// TIA Portal V20 export
FUNCTION_BLOCK "LER_DiagnosticsStatus"   // FB29, LAD
// stored: Access Published, MemoryReserve 100, SetENOAutomatically false
   VAR_INPUT
      devStateHmi_X1 : Array[0..256] of "LAF_typeDevDiagBasic";
      devStateHmi_X2 : Array[0..256] of "LAF_typeDevDiagBasic";
      UnitSelect : Int;
      Reset : Bool;
   END_VAR
   VAR_IN_OUT
      DevState : "LER_DiagnosticsInterface";
   END_VAR
   VAR
      staticCntState : Int := 1;
      staticCntStartState : Int := 1;
      staticCntEndState : Int := 200;
      staticCntDev : Int := 1;
      staticCntHighLimit_X2 : Array[1..15] of Int;
      staticCntLowLimit_X2 : Array[1..15] of Int;
      staticCntHighLimit_X1 : Array[1..15] of Int;
      staticCntLowLimit_X1 : Array[1..15] of Int;
      staticCntModuleState : Int;
      staticDevStateError : Array[0..15] of Bool;
      statiDevStateMove_X1 : Array[0..15] of Int;
      statiDevStateMove_X2 : Array[0..15] of Int;
   END_VAR
   VAR_TEMP
      tempIndex : Int;
   END_VAR
   VAR CONSTANT
      nomal : Word := 16#0009;
   END_VAR
   // staticCntHighLimit_X2[1] := 12;
   // staticCntHighLimit_X2[2] := 14;
   // staticCntHighLimit_X2[3] := 18;
   // staticCntHighLimit_X2[4] := 35;
   // staticCntHighLimit_X2[5] := 38;
   // staticCntHighLimit_X2[6] := 39;
   // staticCntHighLimit_X2[7] := 51;
   // staticCntHighLimit_X2[8] := 53;
   // staticCntLowLimit_X2[2] := 11;
   // staticCntLowLimit_X2[3] := 13;
   // staticCntLowLimit_X2[4] := 17;
   // staticCntLowLimit_X2[5] := 34;
   // staticCntLowLimit_X2[6] := 37;
   // staticCntLowLimit_X2[7] := 38;
   // staticCntLowLimit_X2[8] := 50;
   // staticCntHighLimit_X1[1] := 12;
   // staticCntHighLimit_X1[2] := 14;
   // staticCntHighLimit_X1[3] := 18;
   // staticCntHighLimit_X1[4] := 35;
   // staticCntHighLimit_X1[5] := 38;
   // staticCntHighLimit_X1[6] := 39;
   // staticCntHighLimit_X1[7] := 51;
   // staticCntHighLimit_X1[8] := 53;
   // staticCntLowLimit_X1[2] := 11;
   // staticCntLowLimit_X1[3] := 13;
   // staticCntLowLimit_X1[4] := 17;
   // staticCntLowLimit_X1[5] := 34;
   // staticCntLowLimit_X1[6] := 37;
   // staticCntLowLimit_X1[7] := 38;
   // staticCntLowLimit_X1[8] := 50;
   VAR_TEMP   // added for the SCL form of the ladder/FBD networks
      _w1 : Bool;
      _w2 : Bool;
      _w3 : Bool;
      _w4 : Bool;
      _w5 : Bool;
      _w6 : Bool;
      _w7 : Bool;
      _w8 : Bool;
      _w9 : Bool;
      _w10 : Bool;
      _w11 : Bool;
      _w12 : Bool;
      _w13 : Bool;
      _w14 : Bool;
      _w15 : Bool;
      _w16 : Bool;
   END_VAR
BEGIN

REGION Network 1 (SCL): X1 Port Range
   CASE #UnitSelect OF
       1:  // Unit Reelcut Anode
           #staticCntHighLimit_X1[1] := 0;
           #staticCntHighLimit_X1[2] := 0;
           #staticCntHighLimit_X1[3] := 0;
           #staticCntHighLimit_X1[4] := 18;
           #staticCntHighLimit_X1[5] := 0;
           #staticCntHighLimit_X1[6] := 0;
           #staticCntHighLimit_X1[7] := 41;
           #staticCntHighLimit_X1[8] := 0;
           #staticCntHighLimit_X1[9] := 0;
           #staticCntHighLimit_X1[10] := 0;
           #staticCntHighLimit_X1[11] := 0;
           #staticCntHighLimit_X1[12] := 0;
           #staticCntHighLimit_X1[13] := 0;
           #staticCntHighLimit_X1[14] := 0;
           #staticCntHighLimit_X1[15] := 0;

           #staticCntLowLimit_X1[1] := 0;
           #staticCntLowLimit_X1[2] := 0;
           #staticCntLowLimit_X1[3] := 0;
           #staticCntLowLimit_X1[4] := 18;
           #staticCntLowLimit_X1[5] := 0;
           #staticCntLowLimit_X1[6] := 0;
           #staticCntLowLimit_X1[7] := 39;
           #staticCntLowLimit_X1[8] := 0;
           #staticCntLowLimit_X1[9] := 0;
           #staticCntLowLimit_X1[10] := 0;
           #staticCntLowLimit_X1[11] := 0;
           #staticCntLowLimit_X1[12] := 0;
           #staticCntLowLimit_X1[13] := 0;
           #staticCntLowLimit_X1[14] := 0;
           #staticCntLowLimit_X1[15] := 0;
           ;
       2:  // Unit Reelcut Cathode
           #staticCntHighLimit_X1[1] := 0;
           #staticCntHighLimit_X1[2] := 0;
           #staticCntHighLimit_X1[3] := 0;
           #staticCntHighLimit_X1[4] := 18;
           #staticCntHighLimit_X1[5] := 0;
           #staticCntHighLimit_X1[6] := 0;
           #staticCntHighLimit_X1[7] := 41;
           #staticCntHighLimit_X1[8] := 0;
           #staticCntHighLimit_X1[9] := 0;
           #staticCntHighLimit_X1[10] := 0;
           #staticCntHighLimit_X1[11] := 0;
           #staticCntHighLimit_X1[12] := 0;
           #staticCntHighLimit_X1[13] := 0;
           #staticCntHighLimit_X1[14] := 0;
           #staticCntHighLimit_X1[15] := 0;

           #staticCntLowLimit_X1[1] := 0;
           #staticCntLowLimit_X1[2] := 0;
           #staticCntLowLimit_X1[3] := 0;
           #staticCntLowLimit_X1[4] := 18;
           #staticCntLowLimit_X1[5] := 0;
           #staticCntLowLimit_X1[6] := 0;
           #staticCntLowLimit_X1[7] := 39;
           #staticCntLowLimit_X1[8] := 0;
           #staticCntLowLimit_X1[9] := 0;
           #staticCntLowLimit_X1[10] := 0;
           #staticCntLowLimit_X1[11] := 0;
           #staticCntLowLimit_X1[12] := 0;
           #staticCntLowLimit_X1[13] := 0;
           #staticCntLowLimit_X1[14] := 0;
           #staticCntLowLimit_X1[15] := 0;

       3:  // Unit Stack Anode
           #staticCntHighLimit_X1[1] := 1;
           #staticCntHighLimit_X1[2] := 29;
           #staticCntHighLimit_X1[3] := 41;
           #staticCntHighLimit_X1[4] := 0;
           #staticCntHighLimit_X1[5] := 0;
           #staticCntHighLimit_X1[6] := 0;
           #staticCntHighLimit_X1[7] := 0;
           #staticCntHighLimit_X1[8] := 0;
           #staticCntHighLimit_X1[9] := 0;
           #staticCntHighLimit_X1[10] := 0;
           #staticCntHighLimit_X1[11] := 0;
           #staticCntHighLimit_X1[12] := 0;
           #staticCntHighLimit_X1[13] := 0;
           #staticCntHighLimit_X1[14] := 0;
           #staticCntHighLimit_X1[15] := 0;

           #staticCntLowLimit_X1[1] := 1;
           #staticCntLowLimit_X1[2] := 21;
           #staticCntLowLimit_X1[3] := 41;
           #staticCntLowLimit_X1[4] := 0;
           #staticCntLowLimit_X1[5] := 0;
           #staticCntLowLimit_X1[6] := 0;
           #staticCntLowLimit_X1[7] := 0;
           #staticCntLowLimit_X1[8] := 0;
           #staticCntLowLimit_X1[9] := 0;
           #staticCntLowLimit_X1[10] := 0;
           #staticCntLowLimit_X1[11] := 0;
           #staticCntLowLimit_X1[12] := 0;
           #staticCntLowLimit_X1[13] := 0;
           #staticCntLowLimit_X1[14] := 0;
           #staticCntLowLimit_X1[15] := 0;

       4:  // Unit Stack Cathode
           #staticCntHighLimit_X1[1] := 1;
           #staticCntHighLimit_X1[2] := 29;
           #staticCntHighLimit_X1[3] := 41;
           #staticCntHighLimit_X1[4] := 0;
           #staticCntHighLimit_X1[5] := 0;
           #staticCntHighLimit_X1[6] := 0;
           #staticCntHighLimit_X1[7] := 0;
           #staticCntHighLimit_X1[8] := 0;
           #staticCntHighLimit_X1[9] := 0;
           #staticCntHighLimit_X1[10] := 0;
           #staticCntHighLimit_X1[11] := 0;
           #staticCntHighLimit_X1[12] := 0;
           #staticCntHighLimit_X1[13] := 0;
           #staticCntHighLimit_X1[14] := 0;
           #staticCntHighLimit_X1[15] := 0;

           #staticCntLowLimit_X1[1] := 1;
           #staticCntLowLimit_X1[2] := 21;
           #staticCntLowLimit_X1[3] := 41;
           #staticCntLowLimit_X1[4] := 0;
           #staticCntLowLimit_X1[5] := 0;
           #staticCntLowLimit_X1[6] := 0;
           #staticCntLowLimit_X1[7] := 0;
           #staticCntLowLimit_X1[8] := 0;
           #staticCntLowLimit_X1[9] := 0;
           #staticCntLowLimit_X1[10] := 0;
           #staticCntLowLimit_X1[11] := 0;
           #staticCntLowLimit_X1[12] := 0;
           #staticCntLowLimit_X1[13] := 0;
           #staticCntLowLimit_X1[14] := 0;
           #staticCntLowLimit_X1[15] := 0;

       5:  // Unit Inspection
           #staticCntHighLimit_X1[1] := 0;
           #staticCntHighLimit_X1[2] := 0;
           #staticCntHighLimit_X1[3] := 0;
           #staticCntHighLimit_X1[4] := 64;
           #staticCntHighLimit_X1[5] := 0;
           #staticCntHighLimit_X1[6] := 0;
           #staticCntHighLimit_X1[7] := 0;
           #staticCntHighLimit_X1[8] := 0;
           #staticCntHighLimit_X1[9] := 0;
           #staticCntHighLimit_X1[10] := 0;
           #staticCntHighLimit_X1[11] := 0;
           #staticCntHighLimit_X1[12] := 0;
           #staticCntHighLimit_X1[13] := 243;
           #staticCntHighLimit_X1[14] := 0;
           #staticCntHighLimit_X1[15] := 0;

           #staticCntLowLimit_X1[1] := 0;
           #staticCntLowLimit_X1[2] := 0;
           #staticCntLowLimit_X1[3] := 0;
           #staticCntLowLimit_X1[4] := 61;
           #staticCntLowLimit_X1[5] := 0;
           #staticCntLowLimit_X1[6] := 0;
           #staticCntLowLimit_X1[7] := 0;
           #staticCntLowLimit_X1[8] := 0;
           #staticCntLowLimit_X1[9] := 0;
           #staticCntLowLimit_X1[10] := 0;
           #staticCntLowLimit_X1[11] := 0;
           #staticCntLowLimit_X1[12] := 0;
           #staticCntLowLimit_X1[13] := 241;
           #staticCntLowLimit_X1[14] := 0;
           #staticCntLowLimit_X1[15] := 0;

   END_CASE;
END_REGION

REGION Network 2: X1 Port Data Cnt
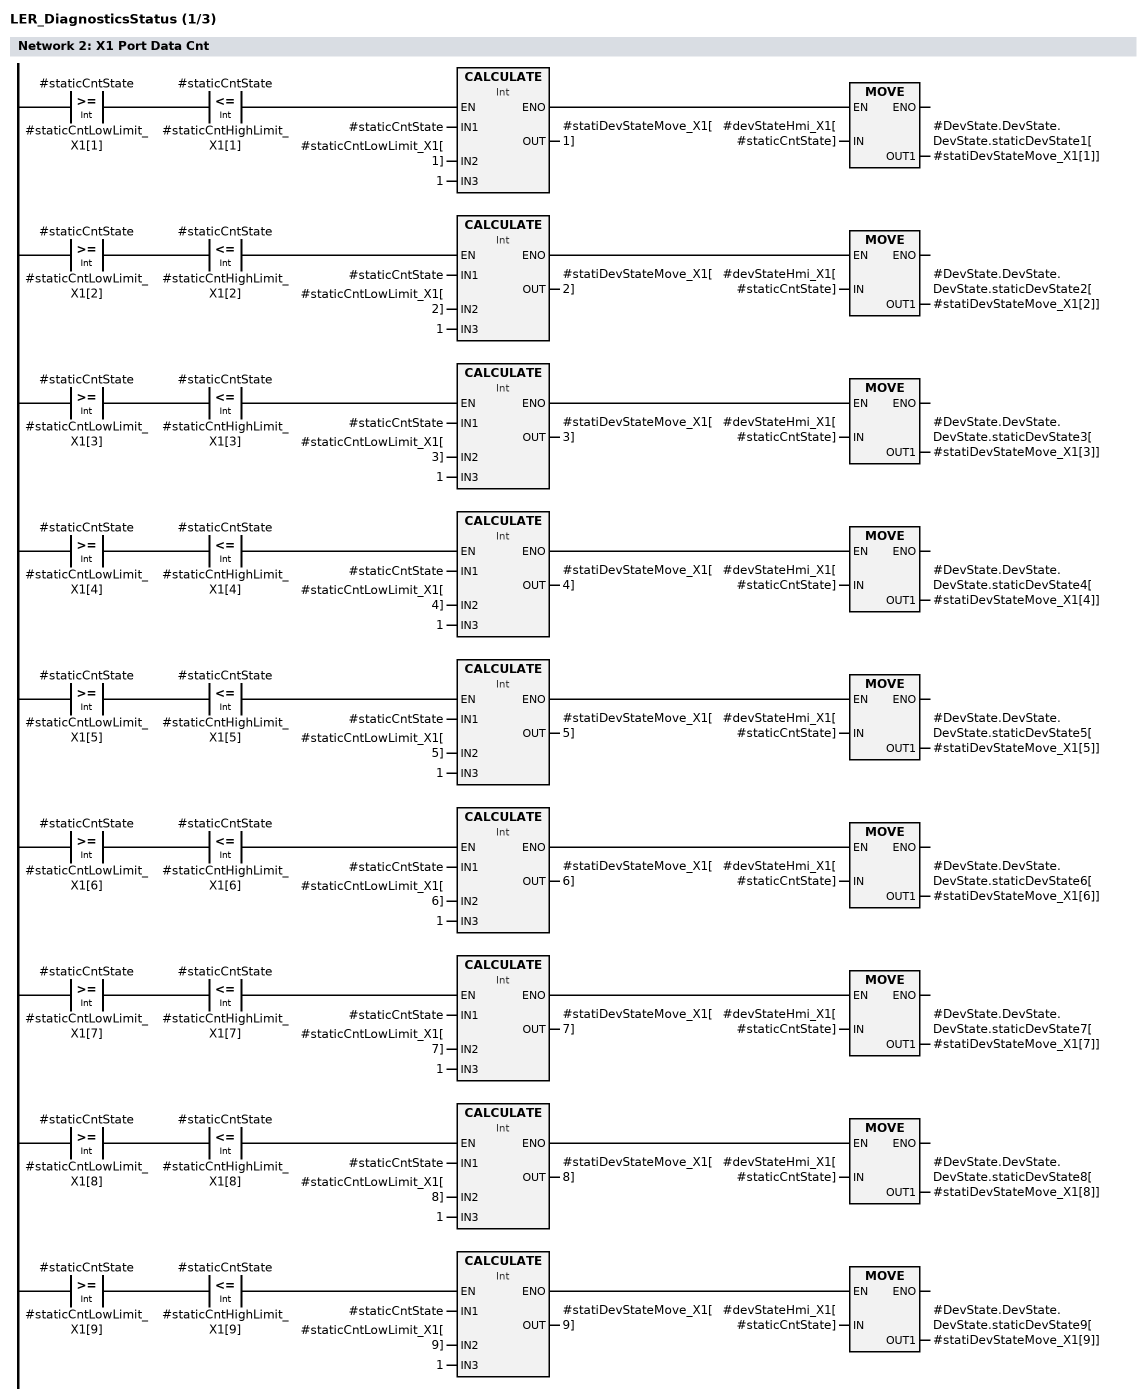
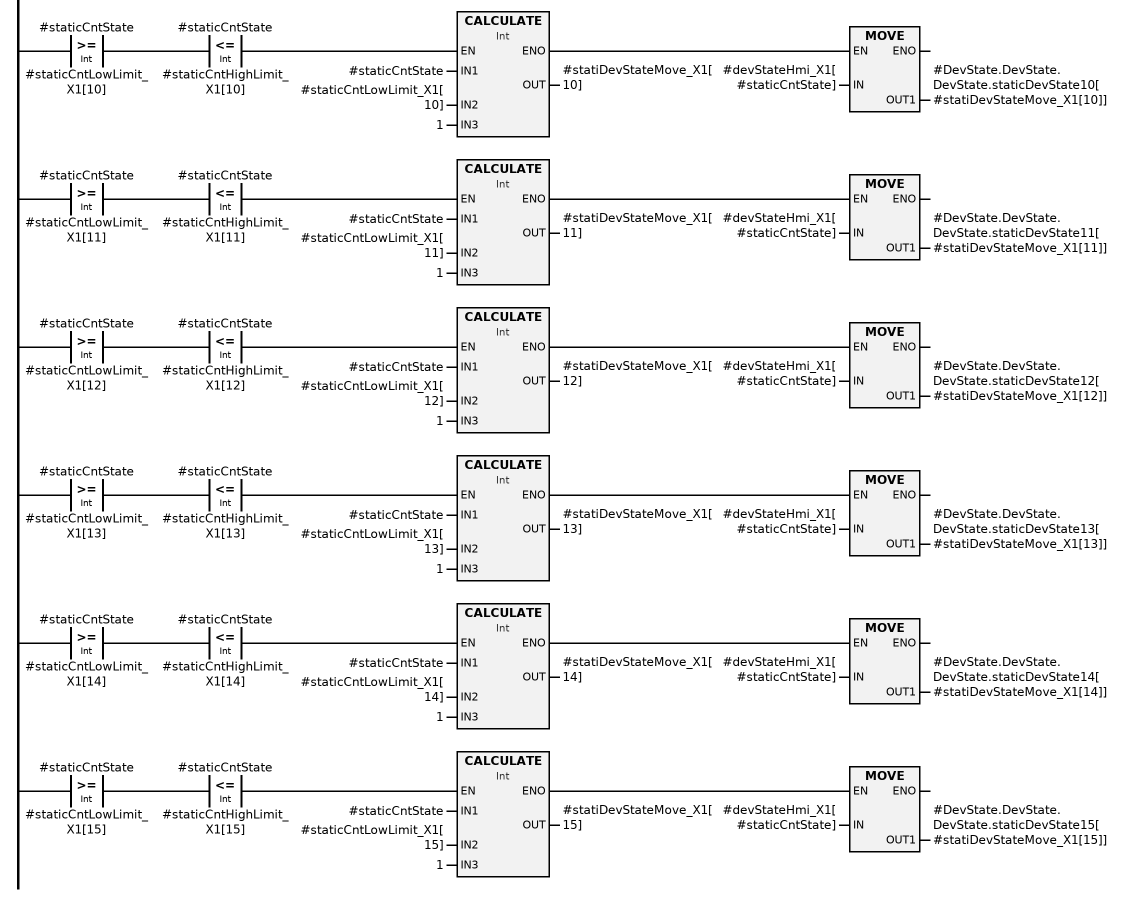
   RUNG wire#powerrail
      { S7_Templates := "SrcType := Int" } GE_Contact(in1 := #staticCntState, in2 := #staticCntLowLimit_X1[1])
      { S7_Templates := "SrcType := Int" } LE_Contact(in1 := #staticCntState, in2 := #staticCntHighLimit_X1[1])
      { S7_Templates := "SrcType := Int"; S7_Expression := "IN1-IN2+IN3" } Calculate(in1 := #staticCntState, in2 := #staticCntLowLimit_X1[1], in3 := 1, out => #statiDevStateMove_X1[1])
      Move(in := #devStateHmi_X1[#staticCntState], out1 => #DevState.DevState.DevState.staticDevState1[#statiDevStateMove_X1[1]])
   END_RUNG
   RUNG wire#powerrail
      { S7_Templates := "SrcType := Int" } GE_Contact(in1 := #staticCntState, in2 := #staticCntLowLimit_X1[2])
      { S7_Templates := "SrcType := Int" } LE_Contact(in1 := #staticCntState, in2 := #staticCntHighLimit_X1[2])
      { S7_Templates := "SrcType := Int"; S7_Expression := "IN1-IN2+IN3" } Calculate(in1 := #staticCntState, in2 := #staticCntLowLimit_X1[2], in3 := 1, out => #statiDevStateMove_X1[2])
      Move(in := #devStateHmi_X1[#staticCntState], out1 => #DevState.DevState.DevState.staticDevState2[#statiDevStateMove_X1[2]])
   END_RUNG
   RUNG wire#powerrail
      { S7_Templates := "SrcType := Int" } GE_Contact(in1 := #staticCntState, in2 := #staticCntLowLimit_X1[3])
      { S7_Templates := "SrcType := Int" } LE_Contact(in1 := #staticCntState, in2 := #staticCntHighLimit_X1[3])
      { S7_Templates := "SrcType := Int"; S7_Expression := "IN1-IN2+IN3" } Calculate(in1 := #staticCntState, in2 := #staticCntLowLimit_X1[3], in3 := 1, out => #statiDevStateMove_X1[3])
      Move(in := #devStateHmi_X1[#staticCntState], out1 => #DevState.DevState.DevState.staticDevState3[#statiDevStateMove_X1[3]])
   END_RUNG
   RUNG wire#powerrail
      { S7_Templates := "SrcType := Int" } GE_Contact(in1 := #staticCntState, in2 := #staticCntLowLimit_X1[4])
      { S7_Templates := "SrcType := Int" } LE_Contact(in1 := #staticCntState, in2 := #staticCntHighLimit_X1[4])
      { S7_Templates := "SrcType := Int"; S7_Expression := "IN1-IN2+IN3" } Calculate(in1 := #staticCntState, in2 := #staticCntLowLimit_X1[4], in3 := 1, out => #statiDevStateMove_X1[4])
      Move(in := #devStateHmi_X1[#staticCntState], out1 => #DevState.DevState.DevState.staticDevState4[#statiDevStateMove_X1[4]])
   END_RUNG
   RUNG wire#powerrail
      { S7_Templates := "SrcType := Int" } GE_Contact(in1 := #staticCntState, in2 := #staticCntLowLimit_X1[5])
      { S7_Templates := "SrcType := Int" } LE_Contact(in1 := #staticCntState, in2 := #staticCntHighLimit_X1[5])
      { S7_Templates := "SrcType := Int"; S7_Expression := "IN1-IN2+IN3" } Calculate(in1 := #staticCntState, in2 := #staticCntLowLimit_X1[5], in3 := 1, out => #statiDevStateMove_X1[5])
      Move(in := #devStateHmi_X1[#staticCntState], out1 => #DevState.DevState.DevState.staticDevState5[#statiDevStateMove_X1[5]])
   END_RUNG
   RUNG wire#powerrail
      { S7_Templates := "SrcType := Int" } GE_Contact(in1 := #staticCntState, in2 := #staticCntLowLimit_X1[6])
      { S7_Templates := "SrcType := Int" } LE_Contact(in1 := #staticCntState, in2 := #staticCntHighLimit_X1[6])
      { S7_Templates := "SrcType := Int"; S7_Expression := "IN1-IN2+IN3" } Calculate(in1 := #staticCntState, in2 := #staticCntLowLimit_X1[6], in3 := 1, out => #statiDevStateMove_X1[6])
      Move(in := #devStateHmi_X1[#staticCntState], out1 => #DevState.DevState.DevState.staticDevState6[#statiDevStateMove_X1[6]])
   END_RUNG
   RUNG wire#powerrail
      { S7_Templates := "SrcType := Int" } GE_Contact(in1 := #staticCntState, in2 := #staticCntLowLimit_X1[7])
      { S7_Templates := "SrcType := Int" } LE_Contact(in1 := #staticCntState, in2 := #staticCntHighLimit_X1[7])
      { S7_Templates := "SrcType := Int"; S7_Expression := "IN1-IN2+IN3" } Calculate(in1 := #staticCntState, in2 := #staticCntLowLimit_X1[7], in3 := 1, out => #statiDevStateMove_X1[7])
      Move(in := #devStateHmi_X1[#staticCntState], out1 => #DevState.DevState.DevState.staticDevState7[#statiDevStateMove_X1[7]])
   END_RUNG
   RUNG wire#powerrail
      { S7_Templates := "SrcType := Int" } GE_Contact(in1 := #staticCntState, in2 := #staticCntLowLimit_X1[8])
      { S7_Templates := "SrcType := Int" } LE_Contact(in1 := #staticCntState, in2 := #staticCntHighLimit_X1[8])
      { S7_Templates := "SrcType := Int"; S7_Expression := "IN1-IN2+IN3" } Calculate(in1 := #staticCntState, in2 := #staticCntLowLimit_X1[8], in3 := 1, out => #statiDevStateMove_X1[8])
      Move(in := #devStateHmi_X1[#staticCntState], out1 => #DevState.DevState.DevState.staticDevState8[#statiDevStateMove_X1[8]])
   END_RUNG
   RUNG wire#powerrail
      { S7_Templates := "SrcType := Int" } GE_Contact(in1 := #staticCntState, in2 := #staticCntLowLimit_X1[9])
      { S7_Templates := "SrcType := Int" } LE_Contact(in1 := #staticCntState, in2 := #staticCntHighLimit_X1[9])
      { S7_Templates := "SrcType := Int"; S7_Expression := "IN1-IN2+IN3" } Calculate(in1 := #staticCntState, in2 := #staticCntLowLimit_X1[9], in3 := 1, out => #statiDevStateMove_X1[9])
      Move(in := #devStateHmi_X1[#staticCntState], out1 => #DevState.DevState.DevState.staticDevState9[#statiDevStateMove_X1[9]])
   END_RUNG
   RUNG wire#powerrail
      { S7_Templates := "SrcType := Int" } GE_Contact(in1 := #staticCntState, in2 := #staticCntLowLimit_X1[10])
      { S7_Templates := "SrcType := Int" } LE_Contact(in1 := #staticCntState, in2 := #staticCntHighLimit_X1[10])
      { S7_Templates := "SrcType := Int"; S7_Expression := "IN1-IN2+IN3" } Calculate(in1 := #staticCntState, in2 := #staticCntLowLimit_X1[10], in3 := 1, out => #statiDevStateMove_X1[10])
      Move(in := #devStateHmi_X1[#staticCntState], out1 => #DevState.DevState.DevState.staticDevState10[#statiDevStateMove_X1[10]])
   END_RUNG
   RUNG wire#powerrail
      { S7_Templates := "SrcType := Int" } GE_Contact(in1 := #staticCntState, in2 := #staticCntLowLimit_X1[11])
      { S7_Templates := "SrcType := Int" } LE_Contact(in1 := #staticCntState, in2 := #staticCntHighLimit_X1[11])
      { S7_Templates := "SrcType := Int"; S7_Expression := "IN1-IN2+IN3" } Calculate(in1 := #staticCntState, in2 := #staticCntLowLimit_X1[11], in3 := 1, out => #statiDevStateMove_X1[11])
      Move(in := #devStateHmi_X1[#staticCntState], out1 => #DevState.DevState.DevState.staticDevState11[#statiDevStateMove_X1[11]])
   END_RUNG
   RUNG wire#powerrail
      { S7_Templates := "SrcType := Int" } GE_Contact(in1 := #staticCntState, in2 := #staticCntLowLimit_X1[12])
      { S7_Templates := "SrcType := Int" } LE_Contact(in1 := #staticCntState, in2 := #staticCntHighLimit_X1[12])
      { S7_Templates := "SrcType := Int"; S7_Expression := "IN1-IN2+IN3" } Calculate(in1 := #staticCntState, in2 := #staticCntLowLimit_X1[12], in3 := 1, out => #statiDevStateMove_X1[12])
      Move(in := #devStateHmi_X1[#staticCntState], out1 => #DevState.DevState.DevState.staticDevState12[#statiDevStateMove_X1[12]])
   END_RUNG
   RUNG wire#powerrail
      { S7_Templates := "SrcType := Int" } GE_Contact(in1 := #staticCntState, in2 := #staticCntLowLimit_X1[13])
      { S7_Templates := "SrcType := Int" } LE_Contact(in1 := #staticCntState, in2 := #staticCntHighLimit_X1[13])
      { S7_Templates := "SrcType := Int"; S7_Expression := "IN1-IN2+IN3" } Calculate(in1 := #staticCntState, in2 := #staticCntLowLimit_X1[13], in3 := 1, out => #statiDevStateMove_X1[13])
      Move(in := #devStateHmi_X1[#staticCntState], out1 => #DevState.DevState.DevState.staticDevState13[#statiDevStateMove_X1[13]])
   END_RUNG
   RUNG wire#powerrail
      { S7_Templates := "SrcType := Int" } GE_Contact(in1 := #staticCntState, in2 := #staticCntLowLimit_X1[14])
      { S7_Templates := "SrcType := Int" } LE_Contact(in1 := #staticCntState, in2 := #staticCntHighLimit_X1[14])
      { S7_Templates := "SrcType := Int"; S7_Expression := "IN1-IN2+IN3" } Calculate(in1 := #staticCntState, in2 := #staticCntLowLimit_X1[14], in3 := 1, out => #statiDevStateMove_X1[14])
      Move(in := #devStateHmi_X1[#staticCntState], out1 => #DevState.DevState.DevState.staticDevState14[#statiDevStateMove_X1[14]])
   END_RUNG
   RUNG wire#powerrail
      { S7_Templates := "SrcType := Int" } GE_Contact(in1 := #staticCntState, in2 := #staticCntLowLimit_X1[15])
      { S7_Templates := "SrcType := Int" } LE_Contact(in1 := #staticCntState, in2 := #staticCntHighLimit_X1[15])
      { S7_Templates := "SrcType := Int"; S7_Expression := "IN1-IN2+IN3" } Calculate(in1 := #staticCntState, in2 := #staticCntLowLimit_X1[15], in3 := 1, out => #statiDevStateMove_X1[15])
      Move(in := #devStateHmi_X1[#staticCntState], out1 => #DevState.DevState.DevState.staticDevState15[#statiDevStateMove_X1[15]])
   END_RUNG
   // the same network as SCL:
   IF (#staticCntState >= #staticCntLowLimit_X1[1]) AND (#staticCntState <= #staticCntHighLimit_X1[1]) THEN
       #statiDevStateMove_X1[1] := #staticCntState-#staticCntLowLimit_X1[1]+1;
       #DevState.DevState.DevState.staticDevState1[#statiDevStateMove_X1[1]] := #devStateHmi_X1[#staticCntState];
   END_IF;
   IF (#staticCntState >= #staticCntLowLimit_X1[2]) AND (#staticCntState <= #staticCntHighLimit_X1[2]) THEN
       #statiDevStateMove_X1[2] := #staticCntState-#staticCntLowLimit_X1[2]+1;
       #DevState.DevState.DevState.staticDevState2[#statiDevStateMove_X1[2]] := #devStateHmi_X1[#staticCntState];
   END_IF;
   IF (#staticCntState >= #staticCntLowLimit_X1[3]) AND (#staticCntState <= #staticCntHighLimit_X1[3]) THEN
       #statiDevStateMove_X1[3] := #staticCntState-#staticCntLowLimit_X1[3]+1;
       #DevState.DevState.DevState.staticDevState3[#statiDevStateMove_X1[3]] := #devStateHmi_X1[#staticCntState];
   END_IF;
   IF (#staticCntState >= #staticCntLowLimit_X1[4]) AND (#staticCntState <= #staticCntHighLimit_X1[4]) THEN
       #statiDevStateMove_X1[4] := #staticCntState-#staticCntLowLimit_X1[4]+1;
       #DevState.DevState.DevState.staticDevState4[#statiDevStateMove_X1[4]] := #devStateHmi_X1[#staticCntState];
   END_IF;
   IF (#staticCntState >= #staticCntLowLimit_X1[5]) AND (#staticCntState <= #staticCntHighLimit_X1[5]) THEN
       #statiDevStateMove_X1[5] := #staticCntState-#staticCntLowLimit_X1[5]+1;
       #DevState.DevState.DevState.staticDevState5[#statiDevStateMove_X1[5]] := #devStateHmi_X1[#staticCntState];
   END_IF;
   IF (#staticCntState >= #staticCntLowLimit_X1[6]) AND (#staticCntState <= #staticCntHighLimit_X1[6]) THEN
       #statiDevStateMove_X1[6] := #staticCntState-#staticCntLowLimit_X1[6]+1;
       #DevState.DevState.DevState.staticDevState6[#statiDevStateMove_X1[6]] := #devStateHmi_X1[#staticCntState];
   END_IF;
   IF (#staticCntState >= #staticCntLowLimit_X1[7]) AND (#staticCntState <= #staticCntHighLimit_X1[7]) THEN
       #statiDevStateMove_X1[7] := #staticCntState-#staticCntLowLimit_X1[7]+1;
       #DevState.DevState.DevState.staticDevState7[#statiDevStateMove_X1[7]] := #devStateHmi_X1[#staticCntState];
   END_IF;
   IF (#staticCntState >= #staticCntLowLimit_X1[8]) AND (#staticCntState <= #staticCntHighLimit_X1[8]) THEN
       #statiDevStateMove_X1[8] := #staticCntState-#staticCntLowLimit_X1[8]+1;
       #DevState.DevState.DevState.staticDevState8[#statiDevStateMove_X1[8]] := #devStateHmi_X1[#staticCntState];
   END_IF;
   IF (#staticCntState >= #staticCntLowLimit_X1[9]) AND (#staticCntState <= #staticCntHighLimit_X1[9]) THEN
       #statiDevStateMove_X1[9] := #staticCntState-#staticCntLowLimit_X1[9]+1;
       #DevState.DevState.DevState.staticDevState9[#statiDevStateMove_X1[9]] := #devStateHmi_X1[#staticCntState];
   END_IF;
   IF (#staticCntState >= #staticCntLowLimit_X1[10]) AND (#staticCntState <= #staticCntHighLimit_X1[10]) THEN
       #statiDevStateMove_X1[10] := #staticCntState-#staticCntLowLimit_X1[10]+1;
       #DevState.DevState.DevState.staticDevState10[#statiDevStateMove_X1[10]] := #devStateHmi_X1[#staticCntState];
   END_IF;
   IF (#staticCntState >= #staticCntLowLimit_X1[11]) AND (#staticCntState <= #staticCntHighLimit_X1[11]) THEN
       #statiDevStateMove_X1[11] := #staticCntState-#staticCntLowLimit_X1[11]+1;
       #DevState.DevState.DevState.staticDevState11[#statiDevStateMove_X1[11]] := #devStateHmi_X1[#staticCntState];
   END_IF;
   IF (#staticCntState >= #staticCntLowLimit_X1[12]) AND (#staticCntState <= #staticCntHighLimit_X1[12]) THEN
       #statiDevStateMove_X1[12] := #staticCntState-#staticCntLowLimit_X1[12]+1;
       #DevState.DevState.DevState.staticDevState12[#statiDevStateMove_X1[12]] := #devStateHmi_X1[#staticCntState];
   END_IF;
   IF (#staticCntState >= #staticCntLowLimit_X1[13]) AND (#staticCntState <= #staticCntHighLimit_X1[13]) THEN
       #statiDevStateMove_X1[13] := #staticCntState-#staticCntLowLimit_X1[13]+1;
       #DevState.DevState.DevState.staticDevState13[#statiDevStateMove_X1[13]] := #devStateHmi_X1[#staticCntState];
   END_IF;
   IF (#staticCntState >= #staticCntLowLimit_X1[14]) AND (#staticCntState <= #staticCntHighLimit_X1[14]) THEN
       #statiDevStateMove_X1[14] := #staticCntState-#staticCntLowLimit_X1[14]+1;
       #DevState.DevState.DevState.staticDevState14[#statiDevStateMove_X1[14]] := #devStateHmi_X1[#staticCntState];
   END_IF;
   IF (#staticCntState >= #staticCntLowLimit_X1[15]) AND (#staticCntState <= #staticCntHighLimit_X1[15]) THEN
       #statiDevStateMove_X1[15] := #staticCntState-#staticCntLowLimit_X1[15]+1;
       #DevState.DevState.DevState.staticDevState15[#statiDevStateMove_X1[15]] := #devStateHmi_X1[#staticCntState];
   END_IF;
END_REGION

REGION Network 3 (SCL): X2 Port Range
   CASE #UnitSelect OF
       1:  // Unit Reelcut Anode
           #staticCntHighLimit_X2[1] := 11;
           #staticCntHighLimit_X2[2] := 22;
           #staticCntHighLimit_X2[3] := 44;
           #staticCntHighLimit_X2[4] := 77;
           #staticCntHighLimit_X2[5] := 83;
           #staticCntHighLimit_X2[6] := 101;
           #staticCntHighLimit_X2[7] := 132;
           #staticCntHighLimit_X2[8] := 142;
           #staticCntHighLimit_X2[9] := 0;
           #staticCntHighLimit_X2[10] := 0;
           #staticCntHighLimit_X2[11] := 0;
           #staticCntHighLimit_X2[12] := 0;
           #staticCntHighLimit_X2[13] := 0;
           #staticCntHighLimit_X2[14] := 0;
           #staticCntHighLimit_X2[15] := 0;

           #staticCntLowLimit_X2[1] := 1;
           #staticCntLowLimit_X2[2] := 21;
           #staticCntLowLimit_X2[3] := 41;
           #staticCntLowLimit_X2[4] := 62;
           #staticCntLowLimit_X2[5] := 81;
           #staticCntLowLimit_X2[6] := 101;
           #staticCntLowLimit_X2[7] := 124;
           #staticCntLowLimit_X2[8] := 141;
           #staticCntLowLimit_X2[9] := 0;
           #staticCntLowLimit_X2[10] := 0;
           #staticCntLowLimit_X2[11] := 0;
           #staticCntLowLimit_X2[12] := 0;
           #staticCntLowLimit_X2[13] := 0;
           #staticCntLowLimit_X2[14] := 0;
           #staticCntLowLimit_X2[15] := 0;
           ;
       2:  // Unit Reelcut Cathode
           #staticCntHighLimit_X2[1] := 11;
           #staticCntHighLimit_X2[2] := 22;
           #staticCntHighLimit_X2[3] := 44;
           #staticCntHighLimit_X2[4] := 77;
           #staticCntHighLimit_X2[5] := 83;
           #staticCntHighLimit_X2[6] := 101;
           #staticCntHighLimit_X2[7] := 132;
           #staticCntHighLimit_X2[8] := 142;
           #staticCntHighLimit_X2[9] := 0;
           #staticCntHighLimit_X2[10] := 0;
           #staticCntHighLimit_X2[11] := 0;
           #staticCntHighLimit_X2[12] := 0;
           #staticCntHighLimit_X2[13] := 0;
           #staticCntHighLimit_X2[14] := 0;
           #staticCntHighLimit_X2[15] := 0;

           #staticCntLowLimit_X2[1] := 1;
           #staticCntLowLimit_X2[2] := 21;
           #staticCntLowLimit_X2[3] := 41;
           #staticCntLowLimit_X2[4] := 62;
           #staticCntLowLimit_X2[5] := 81;
           #staticCntLowLimit_X2[6] := 101;
           #staticCntLowLimit_X2[7] := 124;
           #staticCntLowLimit_X2[8] := 141;
           #staticCntLowLimit_X2[9] := 0;
           #staticCntLowLimit_X2[10] := 0;
           #staticCntLowLimit_X2[11] := 0;
           #staticCntLowLimit_X2[12] := 0;
           #staticCntLowLimit_X2[13] := 0;
           #staticCntLowLimit_X2[14] := 0;
           #staticCntLowLimit_X2[15] := 0;

       3:  // Unit Stack Anode
           #staticCntHighLimit_X2[1] := 2;
           #staticCntHighLimit_X2[2] := 33;
           #staticCntHighLimit_X2[3] := 42;
           #staticCntHighLimit_X2[4] := 68;
           #staticCntHighLimit_X2[5] := 91;
           #staticCntHighLimit_X2[6] := 115;
           #staticCntHighLimit_X2[7] := 133;
           #staticCntHighLimit_X2[8] := 143;
           #staticCntHighLimit_X2[9] := 170;
           #staticCntHighLimit_X2[10] := 0;
           #staticCntHighLimit_X2[11] := 0;
           #staticCntHighLimit_X2[12] := 0;
           #staticCntHighLimit_X2[13] := 0;
           #staticCntHighLimit_X2[14] := 0;
           #staticCntHighLimit_X2[15] := 0;

           #staticCntLowLimit_X2[1] := 2;
           #staticCntLowLimit_X2[2] := 30;
           #staticCntLowLimit_X2[3] := 42;
           #staticCntLowLimit_X2[4] := 61;
           #staticCntLowLimit_X2[5] := 81;
           #staticCntLowLimit_X2[6] := 101;
           #staticCntLowLimit_X2[7] := 121;
           #staticCntLowLimit_X2[8] := 141;
           #staticCntLowLimit_X2[9] := 161;
           #staticCntLowLimit_X2[10] := 0;
           #staticCntLowLimit_X2[11] := 0;
           #staticCntLowLimit_X2[12] := 0;
           #staticCntLowLimit_X2[13] := 0;
           #staticCntLowLimit_X2[14] := 0;
           #staticCntLowLimit_X2[15] := 0;

       4:  // Unit Stack Cathode
           #staticCntHighLimit_X2[1] := 2;
           #staticCntHighLimit_X2[2] := 33;
           #staticCntHighLimit_X2[3] := 42;
           #staticCntHighLimit_X2[4] := 68;
           #staticCntHighLimit_X2[5] := 91;
           #staticCntHighLimit_X2[6] := 115;
           #staticCntHighLimit_X2[7] := 133;
           #staticCntHighLimit_X2[8] := 143;
           #staticCntHighLimit_X2[9] := 170;
           #staticCntHighLimit_X2[10] := 0;
           #staticCntHighLimit_X2[11] := 0;
           #staticCntHighLimit_X2[12] := 0;
           #staticCntHighLimit_X2[13] := 0;
           #staticCntHighLimit_X2[14] := 0;
           #staticCntHighLimit_X2[15] := 0;

           #staticCntLowLimit_X2[1] := 2;
           #staticCntLowLimit_X2[2] := 30;
           #staticCntLowLimit_X2[3] := 42;
           #staticCntLowLimit_X2[4] := 61;
           #staticCntLowLimit_X2[5] := 81;
           #staticCntLowLimit_X2[6] := 101;
           #staticCntLowLimit_X2[7] := 121;
           #staticCntLowLimit_X2[8] := 141;
           #staticCntLowLimit_X2[9] := 161;
           #staticCntLowLimit_X2[10] := 0;
           #staticCntLowLimit_X2[11] := 0;
           #staticCntLowLimit_X2[12] := 0;
           #staticCntLowLimit_X2[13] := 0;
           #staticCntLowLimit_X2[14] := 0;
           #staticCntLowLimit_X2[15] := 0;

       5:  // Unit Inspection
           #staticCntHighLimit_X2[1] := 2;
           #staticCntHighLimit_X2[2] := 25;
           #staticCntHighLimit_X2[3] := 52;
           #staticCntHighLimit_X2[4] := 65;
           #staticCntHighLimit_X2[5] := 97;
           #staticCntHighLimit_X2[6] := 101;
           #staticCntHighLimit_X2[7] := 122;
           #staticCntHighLimit_X2[8] := 146;
           #staticCntHighLimit_X2[9] := 166;
           #staticCntHighLimit_X2[10] := 186;
           #staticCntHighLimit_X2[11] := 204;
           #staticCntHighLimit_X2[12] := 224;
           #staticCntHighLimit_X2[13] := 0;
           #staticCntHighLimit_X2[14] := 0;
           #staticCntHighLimit_X2[15] := 0;

           #staticCntLowLimit_X2[1] := 1;
           #staticCntLowLimit_X2[2] := 21;
           #staticCntLowLimit_X2[3] := 41;
           #staticCntLowLimit_X2[4] := 65;
           #staticCntLowLimit_X2[5] := 81;
           #staticCntLowLimit_X2[6] := 101;
           #staticCntLowLimit_X2[7] := 121;
           #staticCntLowLimit_X2[8] := 141;
           #staticCntLowLimit_X2[9] := 161;
           #staticCntLowLimit_X2[10] := 181;
           #staticCntLowLimit_X2[11] := 201;
           #staticCntLowLimit_X2[12] := 221;
           #staticCntLowLimit_X2[13] := 0;
           #staticCntLowLimit_X2[14] := 0;
           #staticCntLowLimit_X2[15] := 0;

   END_CASE;
END_REGION

REGION Network 4: X2 Port Data Cnt
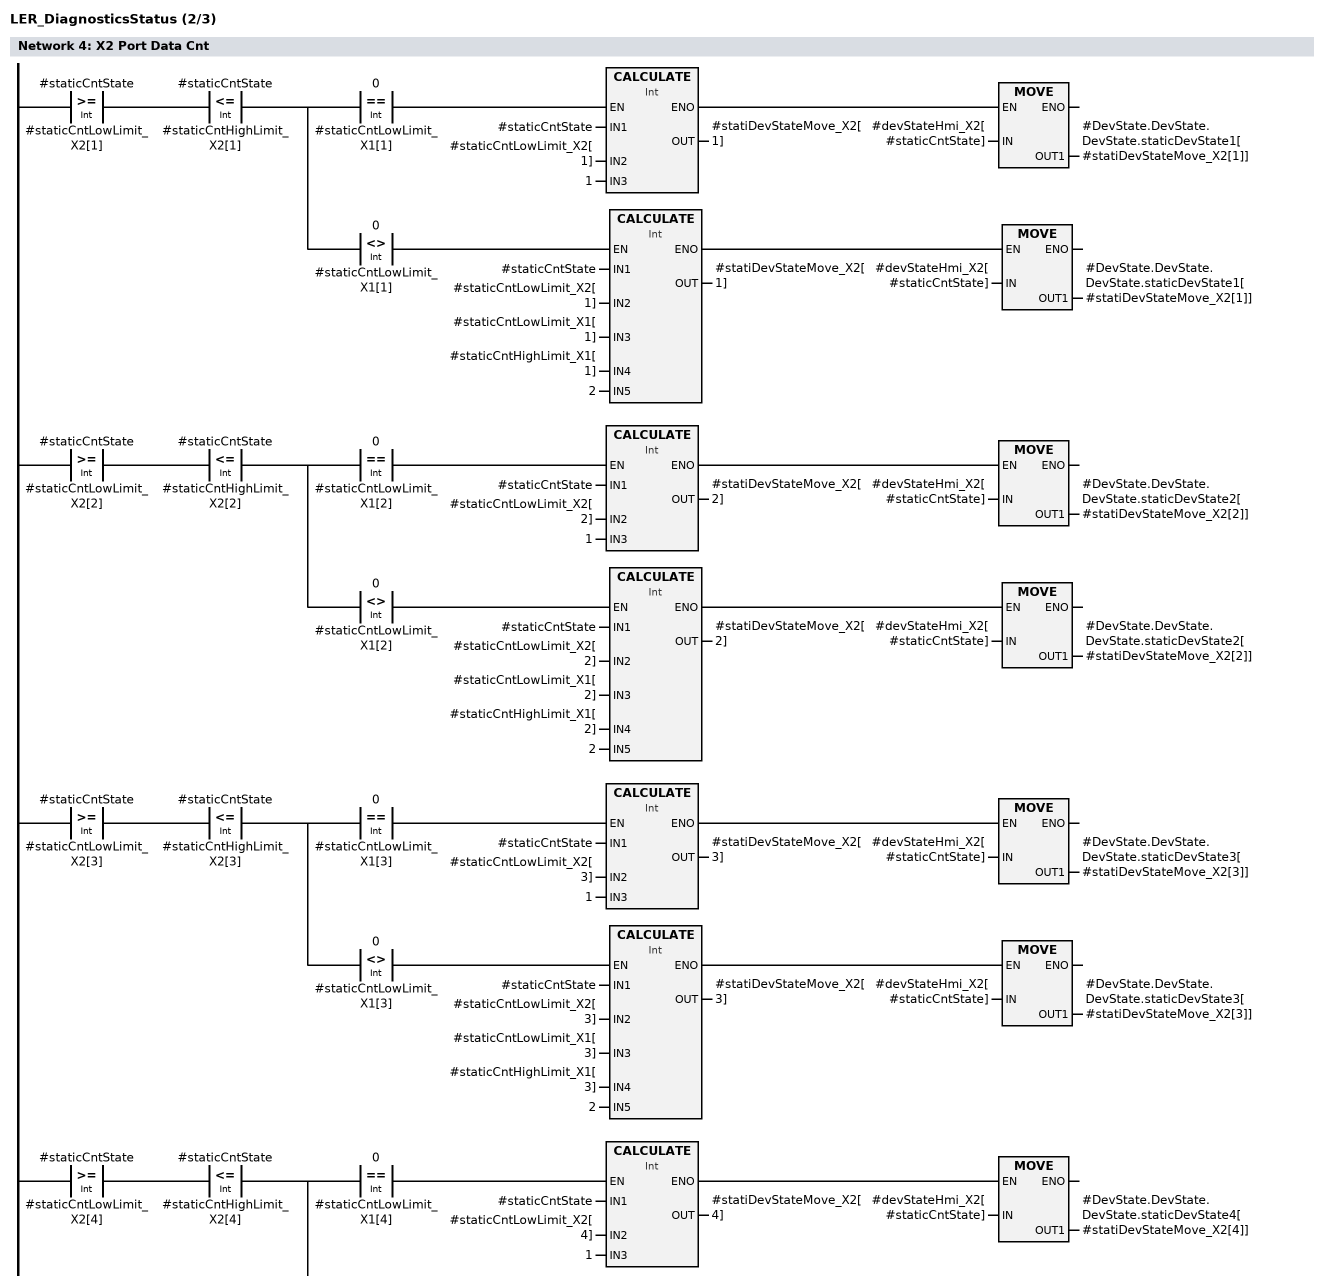
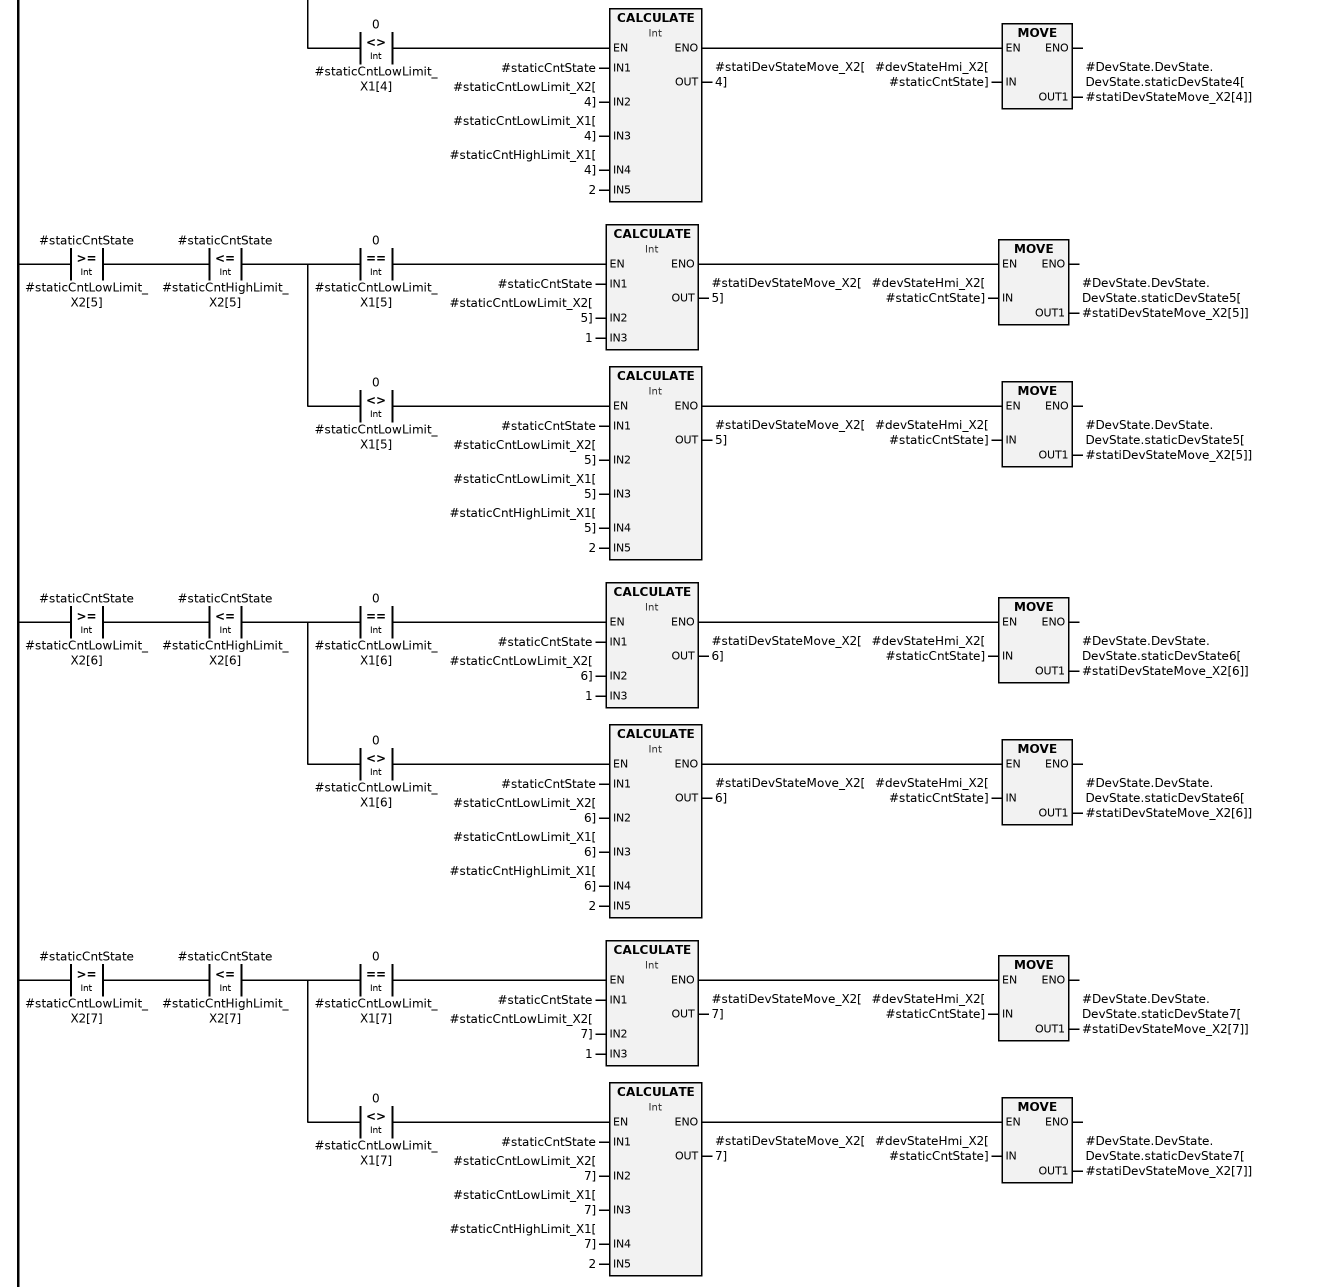
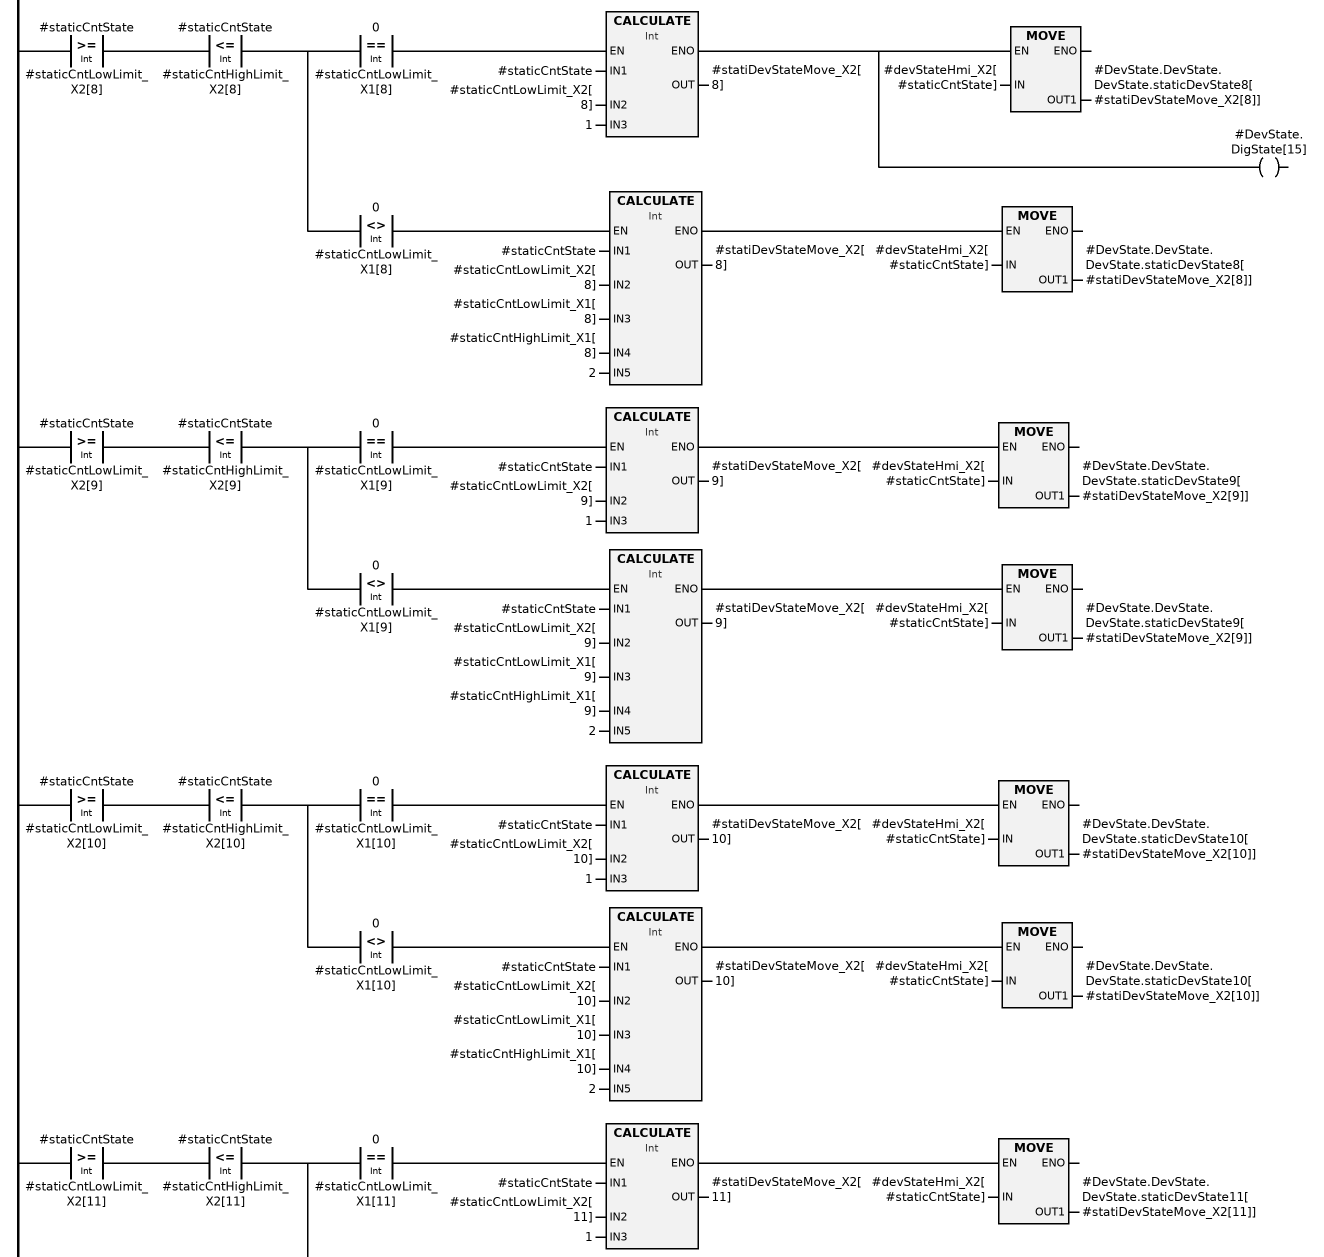
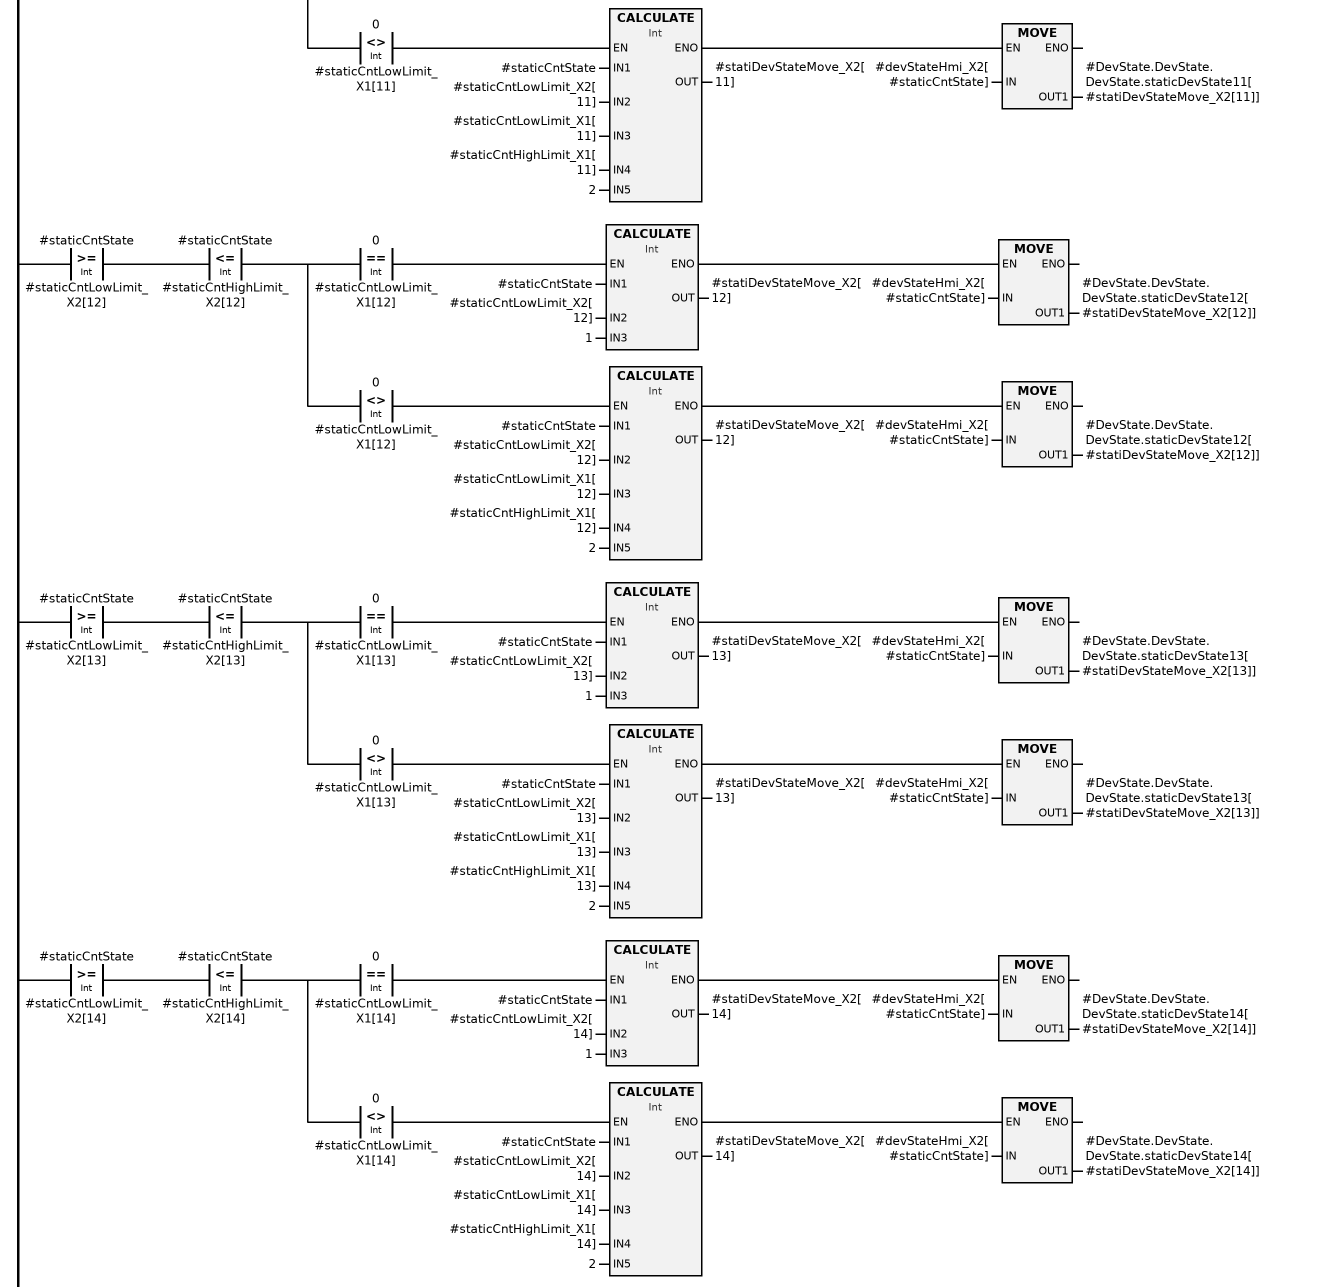
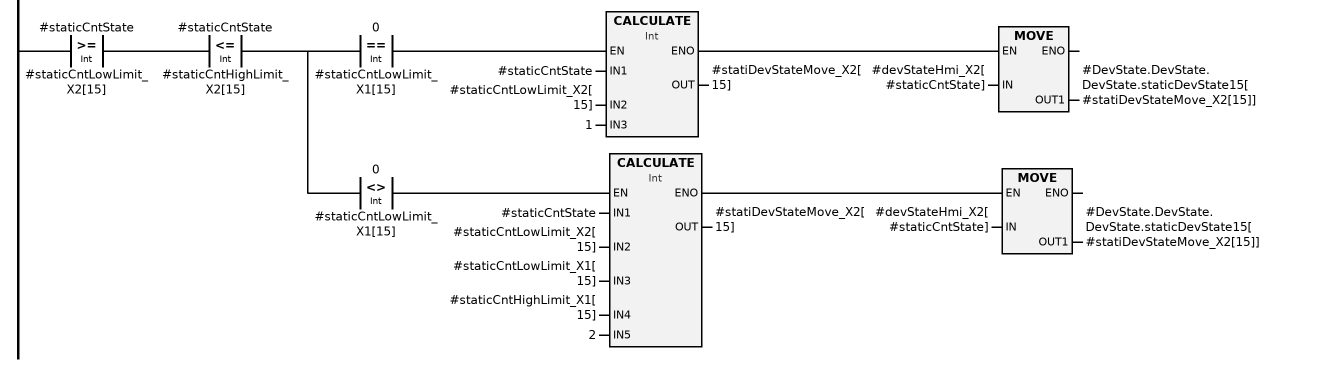
   RUNG wire#powerrail
      { S7_Templates := "SrcType := Int" } GE_Contact(in1 := #staticCntState, in2 := #staticCntLowLimit_X2[1])
      { S7_Templates := "SrcType := Int" } LE_Contact(in1 := #staticCntState, in2 := #staticCntHighLimit_X2[1])
      wire#w1
      { S7_Templates := "SrcType := Int" } EQ_Contact(in1 := 0, in2 := #staticCntLowLimit_X1[1])
      { S7_Templates := "SrcType := Int"; S7_Expression := "IN1-IN2+IN3" } Calculate(in1 := #staticCntState, in2 := #staticCntLowLimit_X2[1], in3 := 1, out => #statiDevStateMove_X2[1])
      Move(in := #devStateHmi_X2[#staticCntState], out1 => #DevState.DevState.DevState.staticDevState1[#statiDevStateMove_X2[1]])
   END_RUNG
   RUNG wire#w1
      { S7_Templates := "SrcType := Int" } NE_Contact(in1 := 0, in2 := #staticCntLowLimit_X1[1])
      { S7_Templates := "SrcType := Int"; S7_Expression := "IN1-IN2+(IN4-IN3+IN5)" } Calculate(in1 := #staticCntState, in2 := #staticCntLowLimit_X2[1], in3 := #staticCntLowLimit_X1[1], in4 := #staticCntHighLimit_X1[1], in5 := 2, out => #statiDevStateMove_X2[1])
      Move(in := #devStateHmi_X2[#staticCntState], out1 => #DevState.DevState.DevState.staticDevState1[#statiDevStateMove_X2[1]])
   END_RUNG
   RUNG wire#powerrail
      { S7_Templates := "SrcType := Int" } GE_Contact(in1 := #staticCntState, in2 := #staticCntLowLimit_X2[2])
      { S7_Templates := "SrcType := Int" } LE_Contact(in1 := #staticCntState, in2 := #staticCntHighLimit_X2[2])
      wire#w2
      { S7_Templates := "SrcType := Int" } EQ_Contact(in1 := 0, in2 := #staticCntLowLimit_X1[2])
      { S7_Templates := "SrcType := Int"; S7_Expression := "IN1-IN2+IN3" } Calculate(in1 := #staticCntState, in2 := #staticCntLowLimit_X2[2], in3 := 1, out => #statiDevStateMove_X2[2])
      Move(in := #devStateHmi_X2[#staticCntState], out1 => #DevState.DevState.DevState.staticDevState2[#statiDevStateMove_X2[2]])
   END_RUNG
   RUNG wire#w2
      { S7_Templates := "SrcType := Int" } NE_Contact(in1 := 0, in2 := #staticCntLowLimit_X1[2])
      { S7_Templates := "SrcType := Int"; S7_Expression := "IN1-IN2+(IN4-IN3+IN5)" } Calculate(in1 := #staticCntState, in2 := #staticCntLowLimit_X2[2], in3 := #staticCntLowLimit_X1[2], in4 := #staticCntHighLimit_X1[2], in5 := 2, out => #statiDevStateMove_X2[2])
      Move(in := #devStateHmi_X2[#staticCntState], out1 => #DevState.DevState.DevState.staticDevState2[#statiDevStateMove_X2[2]])
   END_RUNG
   RUNG wire#powerrail
      { S7_Templates := "SrcType := Int" } GE_Contact(in1 := #staticCntState, in2 := #staticCntLowLimit_X2[3])
      { S7_Templates := "SrcType := Int" } LE_Contact(in1 := #staticCntState, in2 := #staticCntHighLimit_X2[3])
      wire#w3
      { S7_Templates := "SrcType := Int" } EQ_Contact(in1 := 0, in2 := #staticCntLowLimit_X1[3])
      { S7_Templates := "SrcType := Int"; S7_Expression := "IN1-IN2+IN3" } Calculate(in1 := #staticCntState, in2 := #staticCntLowLimit_X2[3], in3 := 1, out => #statiDevStateMove_X2[3])
      Move(in := #devStateHmi_X2[#staticCntState], out1 => #DevState.DevState.DevState.staticDevState3[#statiDevStateMove_X2[3]])
   END_RUNG
   RUNG wire#w3
      { S7_Templates := "SrcType := Int" } NE_Contact(in1 := 0, in2 := #staticCntLowLimit_X1[3])
      { S7_Templates := "SrcType := Int"; S7_Expression := "IN1-IN2+(IN4-IN3+IN5)" } Calculate(in1 := #staticCntState, in2 := #staticCntLowLimit_X2[3], in3 := #staticCntLowLimit_X1[3], in4 := #staticCntHighLimit_X1[3], in5 := 2, out => #statiDevStateMove_X2[3])
      Move(in := #devStateHmi_X2[#staticCntState], out1 => #DevState.DevState.DevState.staticDevState3[#statiDevStateMove_X2[3]])
   END_RUNG
   RUNG wire#powerrail
      { S7_Templates := "SrcType := Int" } GE_Contact(in1 := #staticCntState, in2 := #staticCntLowLimit_X2[4])
      { S7_Templates := "SrcType := Int" } LE_Contact(in1 := #staticCntState, in2 := #staticCntHighLimit_X2[4])
      wire#w4
      { S7_Templates := "SrcType := Int" } EQ_Contact(in1 := 0, in2 := #staticCntLowLimit_X1[4])
      { S7_Templates := "SrcType := Int"; S7_Expression := "IN1-IN2+IN3" } Calculate(in1 := #staticCntState, in2 := #staticCntLowLimit_X2[4], in3 := 1, out => #statiDevStateMove_X2[4])
      Move(in := #devStateHmi_X2[#staticCntState], out1 => #DevState.DevState.DevState.staticDevState4[#statiDevStateMove_X2[4]])
   END_RUNG
   RUNG wire#w4
      { S7_Templates := "SrcType := Int" } NE_Contact(in1 := 0, in2 := #staticCntLowLimit_X1[4])
      { S7_Templates := "SrcType := Int"; S7_Expression := "IN1-IN2+(IN4-IN3+IN5)" } Calculate(in1 := #staticCntState, in2 := #staticCntLowLimit_X2[4], in3 := #staticCntLowLimit_X1[4], in4 := #staticCntHighLimit_X1[4], in5 := 2, out => #statiDevStateMove_X2[4])
      Move(in := #devStateHmi_X2[#staticCntState], out1 => #DevState.DevState.DevState.staticDevState4[#statiDevStateMove_X2[4]])
   END_RUNG
   RUNG wire#powerrail
      { S7_Templates := "SrcType := Int" } GE_Contact(in1 := #staticCntState, in2 := #staticCntLowLimit_X2[5])
      { S7_Templates := "SrcType := Int" } LE_Contact(in1 := #staticCntState, in2 := #staticCntHighLimit_X2[5])
      wire#w5
      { S7_Templates := "SrcType := Int" } EQ_Contact(in1 := 0, in2 := #staticCntLowLimit_X1[5])
      { S7_Templates := "SrcType := Int"; S7_Expression := "IN1-IN2+IN3" } Calculate(in1 := #staticCntState, in2 := #staticCntLowLimit_X2[5], in3 := 1, out => #statiDevStateMove_X2[5])
      Move(in := #devStateHmi_X2[#staticCntState], out1 => #DevState.DevState.DevState.staticDevState5[#statiDevStateMove_X2[5]])
   END_RUNG
   RUNG wire#w5
      { S7_Templates := "SrcType := Int" } NE_Contact(in1 := 0, in2 := #staticCntLowLimit_X1[5])
      { S7_Templates := "SrcType := Int"; S7_Expression := "IN1-IN2+(IN4-IN3+IN5)" } Calculate(in1 := #staticCntState, in2 := #staticCntLowLimit_X2[5], in3 := #staticCntLowLimit_X1[5], in4 := #staticCntHighLimit_X1[5], in5 := 2, out => #statiDevStateMove_X2[5])
      Move(in := #devStateHmi_X2[#staticCntState], out1 => #DevState.DevState.DevState.staticDevState5[#statiDevStateMove_X2[5]])
   END_RUNG
   RUNG wire#powerrail
      { S7_Templates := "SrcType := Int" } GE_Contact(in1 := #staticCntState, in2 := #staticCntLowLimit_X2[6])
      { S7_Templates := "SrcType := Int" } LE_Contact(in1 := #staticCntState, in2 := #staticCntHighLimit_X2[6])
      wire#w6
      { S7_Templates := "SrcType := Int" } EQ_Contact(in1 := 0, in2 := #staticCntLowLimit_X1[6])
      { S7_Templates := "SrcType := Int"; S7_Expression := "IN1-IN2+IN3" } Calculate(in1 := #staticCntState, in2 := #staticCntLowLimit_X2[6], in3 := 1, out => #statiDevStateMove_X2[6])
      Move(in := #devStateHmi_X2[#staticCntState], out1 => #DevState.DevState.DevState.staticDevState6[#statiDevStateMove_X2[6]])
   END_RUNG
   RUNG wire#w6
      { S7_Templates := "SrcType := Int" } NE_Contact(in1 := 0, in2 := #staticCntLowLimit_X1[6])
      { S7_Templates := "SrcType := Int"; S7_Expression := "IN1-IN2+(IN4-IN3+IN5)" } Calculate(in1 := #staticCntState, in2 := #staticCntLowLimit_X2[6], in3 := #staticCntLowLimit_X1[6], in4 := #staticCntHighLimit_X1[6], in5 := 2, out => #statiDevStateMove_X2[6])
      Move(in := #devStateHmi_X2[#staticCntState], out1 => #DevState.DevState.DevState.staticDevState6[#statiDevStateMove_X2[6]])
   END_RUNG
   RUNG wire#powerrail
      { S7_Templates := "SrcType := Int" } GE_Contact(in1 := #staticCntState, in2 := #staticCntLowLimit_X2[7])
      { S7_Templates := "SrcType := Int" } LE_Contact(in1 := #staticCntState, in2 := #staticCntHighLimit_X2[7])
      wire#w7
      { S7_Templates := "SrcType := Int" } EQ_Contact(in1 := 0, in2 := #staticCntLowLimit_X1[7])
      { S7_Templates := "SrcType := Int"; S7_Expression := "IN1-IN2+IN3" } Calculate(in1 := #staticCntState, in2 := #staticCntLowLimit_X2[7], in3 := 1, out => #statiDevStateMove_X2[7])
      Move(in := #devStateHmi_X2[#staticCntState], out1 => #DevState.DevState.DevState.staticDevState7[#statiDevStateMove_X2[7]])
   END_RUNG
   RUNG wire#w7
      { S7_Templates := "SrcType := Int" } NE_Contact(in1 := 0, in2 := #staticCntLowLimit_X1[7])
      { S7_Templates := "SrcType := Int"; S7_Expression := "IN1-IN2+(IN4-IN3+IN5)" } Calculate(in1 := #staticCntState, in2 := #staticCntLowLimit_X2[7], in3 := #staticCntLowLimit_X1[7], in4 := #staticCntHighLimit_X1[7], in5 := 2, out => #statiDevStateMove_X2[7])
      Move(in := #devStateHmi_X2[#staticCntState], out1 => #DevState.DevState.DevState.staticDevState7[#statiDevStateMove_X2[7]])
   END_RUNG
   RUNG wire#powerrail
      { S7_Templates := "SrcType := Int" } GE_Contact(in1 := #staticCntState, in2 := #staticCntLowLimit_X2[8])
      { S7_Templates := "SrcType := Int" } LE_Contact(in1 := #staticCntState, in2 := #staticCntHighLimit_X2[8])
      wire#w8
      { S7_Templates := "SrcType := Int" } EQ_Contact(in1 := 0, in2 := #staticCntLowLimit_X1[8])
      { S7_Templates := "SrcType := Int"; S7_Expression := "IN1-IN2+IN3" } Calculate(in1 := #staticCntState, in2 := #staticCntLowLimit_X2[8], in3 := 1, out => #statiDevStateMove_X2[8])
      wire#w9
      Move(in := #devStateHmi_X2[#staticCntState], out1 => #DevState.DevState.DevState.staticDevState8[#statiDevStateMove_X2[8]])
   END_RUNG
   RUNG wire#w9
      Coil( #DevState.DigState[15] )
   END_RUNG
   RUNG wire#w8
      { S7_Templates := "SrcType := Int" } NE_Contact(in1 := 0, in2 := #staticCntLowLimit_X1[8])
      { S7_Templates := "SrcType := Int"; S7_Expression := "IN1-IN2+(IN4-IN3+IN5)" } Calculate(in1 := #staticCntState, in2 := #staticCntLowLimit_X2[8], in3 := #staticCntLowLimit_X1[8], in4 := #staticCntHighLimit_X1[8], in5 := 2, out => #statiDevStateMove_X2[8])
      Move(in := #devStateHmi_X2[#staticCntState], out1 => #DevState.DevState.DevState.staticDevState8[#statiDevStateMove_X2[8]])
   END_RUNG
   RUNG wire#powerrail
      { S7_Templates := "SrcType := Int" } GE_Contact(in1 := #staticCntState, in2 := #staticCntLowLimit_X2[9])
      { S7_Templates := "SrcType := Int" } LE_Contact(in1 := #staticCntState, in2 := #staticCntHighLimit_X2[9])
      wire#w10
      { S7_Templates := "SrcType := Int" } EQ_Contact(in1 := 0, in2 := #staticCntLowLimit_X1[9])
      { S7_Templates := "SrcType := Int"; S7_Expression := "IN1-IN2+IN3" } Calculate(in1 := #staticCntState, in2 := #staticCntLowLimit_X2[9], in3 := 1, out => #statiDevStateMove_X2[9])
      Move(in := #devStateHmi_X2[#staticCntState], out1 => #DevState.DevState.DevState.staticDevState9[#statiDevStateMove_X2[9]])
   END_RUNG
   RUNG wire#w10
      { S7_Templates := "SrcType := Int" } NE_Contact(in1 := 0, in2 := #staticCntLowLimit_X1[9])
      { S7_Templates := "SrcType := Int"; S7_Expression := "IN1-IN2+(IN4-IN3+IN5)" } Calculate(in1 := #staticCntState, in2 := #staticCntLowLimit_X2[9], in3 := #staticCntLowLimit_X1[9], in4 := #staticCntHighLimit_X1[9], in5 := 2, out => #statiDevStateMove_X2[9])
      Move(in := #devStateHmi_X2[#staticCntState], out1 => #DevState.DevState.DevState.staticDevState9[#statiDevStateMove_X2[9]])
   END_RUNG
   RUNG wire#powerrail
      { S7_Templates := "SrcType := Int" } GE_Contact(in1 := #staticCntState, in2 := #staticCntLowLimit_X2[10])
      { S7_Templates := "SrcType := Int" } LE_Contact(in1 := #staticCntState, in2 := #staticCntHighLimit_X2[10])
      wire#w11
      { S7_Templates := "SrcType := Int" } EQ_Contact(in1 := 0, in2 := #staticCntLowLimit_X1[10])
      { S7_Templates := "SrcType := Int"; S7_Expression := "IN1-IN2+IN3" } Calculate(in1 := #staticCntState, in2 := #staticCntLowLimit_X2[10], in3 := 1, out => #statiDevStateMove_X2[10])
      Move(in := #devStateHmi_X2[#staticCntState], out1 => #DevState.DevState.DevState.staticDevState10[#statiDevStateMove_X2[10]])
   END_RUNG
   RUNG wire#w11
      { S7_Templates := "SrcType := Int" } NE_Contact(in1 := 0, in2 := #staticCntLowLimit_X1[10])
      { S7_Templates := "SrcType := Int"; S7_Expression := "IN1-IN2+(IN4-IN3+IN5)" } Calculate(in1 := #staticCntState, in2 := #staticCntLowLimit_X2[10], in3 := #staticCntLowLimit_X1[10], in4 := #staticCntHighLimit_X1[10], in5 := 2, out => #statiDevStateMove_X2[10])
      Move(in := #devStateHmi_X2[#staticCntState], out1 => #DevState.DevState.DevState.staticDevState10[#statiDevStateMove_X2[10]])
   END_RUNG
   RUNG wire#powerrail
      { S7_Templates := "SrcType := Int" } GE_Contact(in1 := #staticCntState, in2 := #staticCntLowLimit_X2[11])
      { S7_Templates := "SrcType := Int" } LE_Contact(in1 := #staticCntState, in2 := #staticCntHighLimit_X2[11])
      wire#w12
      { S7_Templates := "SrcType := Int" } EQ_Contact(in1 := 0, in2 := #staticCntLowLimit_X1[11])
      { S7_Templates := "SrcType := Int"; S7_Expression := "IN1-IN2+IN3" } Calculate(in1 := #staticCntState, in2 := #staticCntLowLimit_X2[11], in3 := 1, out => #statiDevStateMove_X2[11])
      Move(in := #devStateHmi_X2[#staticCntState], out1 => #DevState.DevState.DevState.staticDevState11[#statiDevStateMove_X2[11]])
   END_RUNG
   RUNG wire#w12
      { S7_Templates := "SrcType := Int" } NE_Contact(in1 := 0, in2 := #staticCntLowLimit_X1[11])
      { S7_Templates := "SrcType := Int"; S7_Expression := "IN1-IN2+(IN4-IN3+IN5)" } Calculate(in1 := #staticCntState, in2 := #staticCntLowLimit_X2[11], in3 := #staticCntLowLimit_X1[11], in4 := #staticCntHighLimit_X1[11], in5 := 2, out => #statiDevStateMove_X2[11])
      Move(in := #devStateHmi_X2[#staticCntState], out1 => #DevState.DevState.DevState.staticDevState11[#statiDevStateMove_X2[11]])
   END_RUNG
   RUNG wire#powerrail
      { S7_Templates := "SrcType := Int" } GE_Contact(in1 := #staticCntState, in2 := #staticCntLowLimit_X2[12])
      { S7_Templates := "SrcType := Int" } LE_Contact(in1 := #staticCntState, in2 := #staticCntHighLimit_X2[12])
      wire#w13
      { S7_Templates := "SrcType := Int" } EQ_Contact(in1 := 0, in2 := #staticCntLowLimit_X1[12])
      { S7_Templates := "SrcType := Int"; S7_Expression := "IN1-IN2+IN3" } Calculate(in1 := #staticCntState, in2 := #staticCntLowLimit_X2[12], in3 := 1, out => #statiDevStateMove_X2[12])
      Move(in := #devStateHmi_X2[#staticCntState], out1 => #DevState.DevState.DevState.staticDevState12[#statiDevStateMove_X2[12]])
   END_RUNG
   RUNG wire#w13
      { S7_Templates := "SrcType := Int" } NE_Contact(in1 := 0, in2 := #staticCntLowLimit_X1[12])
      { S7_Templates := "SrcType := Int"; S7_Expression := "IN1-IN2+(IN4-IN3+IN5)" } Calculate(in1 := #staticCntState, in2 := #staticCntLowLimit_X2[12], in3 := #staticCntLowLimit_X1[12], in4 := #staticCntHighLimit_X1[12], in5 := 2, out => #statiDevStateMove_X2[12])
      Move(in := #devStateHmi_X2[#staticCntState], out1 => #DevState.DevState.DevState.staticDevState12[#statiDevStateMove_X2[12]])
   END_RUNG
   RUNG wire#powerrail
      { S7_Templates := "SrcType := Int" } GE_Contact(in1 := #staticCntState, in2 := #staticCntLowLimit_X2[13])
      { S7_Templates := "SrcType := Int" } LE_Contact(in1 := #staticCntState, in2 := #staticCntHighLimit_X2[13])
      wire#w14
      { S7_Templates := "SrcType := Int" } EQ_Contact(in1 := 0, in2 := #staticCntLowLimit_X1[13])
      { S7_Templates := "SrcType := Int"; S7_Expression := "IN1-IN2+IN3" } Calculate(in1 := #staticCntState, in2 := #staticCntLowLimit_X2[13], in3 := 1, out => #statiDevStateMove_X2[13])
      Move(in := #devStateHmi_X2[#staticCntState], out1 => #DevState.DevState.DevState.staticDevState13[#statiDevStateMove_X2[13]])
   END_RUNG
   RUNG wire#w14
      { S7_Templates := "SrcType := Int" } NE_Contact(in1 := 0, in2 := #staticCntLowLimit_X1[13])
      { S7_Templates := "SrcType := Int"; S7_Expression := "IN1-IN2+(IN4-IN3+IN5)" } Calculate(in1 := #staticCntState, in2 := #staticCntLowLimit_X2[13], in3 := #staticCntLowLimit_X1[13], in4 := #staticCntHighLimit_X1[13], in5 := 2, out => #statiDevStateMove_X2[13])
      Move(in := #devStateHmi_X2[#staticCntState], out1 => #DevState.DevState.DevState.staticDevState13[#statiDevStateMove_X2[13]])
   END_RUNG
   RUNG wire#powerrail
      { S7_Templates := "SrcType := Int" } GE_Contact(in1 := #staticCntState, in2 := #staticCntLowLimit_X2[14])
      { S7_Templates := "SrcType := Int" } LE_Contact(in1 := #staticCntState, in2 := #staticCntHighLimit_X2[14])
      wire#w15
      { S7_Templates := "SrcType := Int" } EQ_Contact(in1 := 0, in2 := #staticCntLowLimit_X1[14])
      { S7_Templates := "SrcType := Int"; S7_Expression := "IN1-IN2+IN3" } Calculate(in1 := #staticCntState, in2 := #staticCntLowLimit_X2[14], in3 := 1, out => #statiDevStateMove_X2[14])
      Move(in := #devStateHmi_X2[#staticCntState], out1 => #DevState.DevState.DevState.staticDevState14[#statiDevStateMove_X2[14]])
   END_RUNG
   RUNG wire#w15
      { S7_Templates := "SrcType := Int" } NE_Contact(in1 := 0, in2 := #staticCntLowLimit_X1[14])
      { S7_Templates := "SrcType := Int"; S7_Expression := "IN1-IN2+(IN4-IN3+IN5)" } Calculate(in1 := #staticCntState, in2 := #staticCntLowLimit_X2[14], in3 := #staticCntLowLimit_X1[14], in4 := #staticCntHighLimit_X1[14], in5 := 2, out => #statiDevStateMove_X2[14])
      Move(in := #devStateHmi_X2[#staticCntState], out1 => #DevState.DevState.DevState.staticDevState14[#statiDevStateMove_X2[14]])
   END_RUNG
   RUNG wire#powerrail
      { S7_Templates := "SrcType := Int" } GE_Contact(in1 := #staticCntState, in2 := #staticCntLowLimit_X2[15])
      { S7_Templates := "SrcType := Int" } LE_Contact(in1 := #staticCntState, in2 := #staticCntHighLimit_X2[15])
      wire#w16
      { S7_Templates := "SrcType := Int" } EQ_Contact(in1 := 0, in2 := #staticCntLowLimit_X1[15])
      { S7_Templates := "SrcType := Int"; S7_Expression := "IN1-IN2+IN3" } Calculate(in1 := #staticCntState, in2 := #staticCntLowLimit_X2[15], in3 := 1, out => #statiDevStateMove_X2[15])
      Move(in := #devStateHmi_X2[#staticCntState], out1 => #DevState.DevState.DevState.staticDevState15[#statiDevStateMove_X2[15]])
   END_RUNG
   RUNG wire#w16
      { S7_Templates := "SrcType := Int" } NE_Contact(in1 := 0, in2 := #staticCntLowLimit_X1[15])
      { S7_Templates := "SrcType := Int"; S7_Expression := "IN1-IN2+(IN4-IN3+IN5)" } Calculate(in1 := #staticCntState, in2 := #staticCntLowLimit_X2[15], in3 := #staticCntLowLimit_X1[15], in4 := #staticCntHighLimit_X1[15], in5 := 2, out => #statiDevStateMove_X2[15])
      Move(in := #devStateHmi_X2[#staticCntState], out1 => #DevState.DevState.DevState.staticDevState15[#statiDevStateMove_X2[15]])
   END_RUNG
   // the same network as SCL:
   #_w1 := (#staticCntState >= #staticCntLowLimit_X2[1]) AND (#staticCntState <= #staticCntHighLimit_X2[1]);
   IF #_w1 AND (0 = #staticCntLowLimit_X1[1]) THEN
       #statiDevStateMove_X2[1] := #staticCntState-#staticCntLowLimit_X2[1]+1;
       #DevState.DevState.DevState.staticDevState1[#statiDevStateMove_X2[1]] := #devStateHmi_X2[#staticCntState];
   END_IF;
   IF #_w1 AND (0 <> #staticCntLowLimit_X1[1]) THEN
       #statiDevStateMove_X2[1] := #staticCntState-#staticCntLowLimit_X2[1]+(#staticCntHighLimit_X1[1]-#staticCntLowLimit_X1[1]+2);
       #DevState.DevState.DevState.staticDevState1[#statiDevStateMove_X2[1]] := #devStateHmi_X2[#staticCntState];
   END_IF;
   #_w2 := (#staticCntState >= #staticCntLowLimit_X2[2]) AND (#staticCntState <= #staticCntHighLimit_X2[2]);
   IF #_w2 AND (0 = #staticCntLowLimit_X1[2]) THEN
       #statiDevStateMove_X2[2] := #staticCntState-#staticCntLowLimit_X2[2]+1;
       #DevState.DevState.DevState.staticDevState2[#statiDevStateMove_X2[2]] := #devStateHmi_X2[#staticCntState];
   END_IF;
   IF #_w2 AND (0 <> #staticCntLowLimit_X1[2]) THEN
       #statiDevStateMove_X2[2] := #staticCntState-#staticCntLowLimit_X2[2]+(#staticCntHighLimit_X1[2]-#staticCntLowLimit_X1[2]+2);
       #DevState.DevState.DevState.staticDevState2[#statiDevStateMove_X2[2]] := #devStateHmi_X2[#staticCntState];
   END_IF;
   #_w3 := (#staticCntState >= #staticCntLowLimit_X2[3]) AND (#staticCntState <= #staticCntHighLimit_X2[3]);
   IF #_w3 AND (0 = #staticCntLowLimit_X1[3]) THEN
       #statiDevStateMove_X2[3] := #staticCntState-#staticCntLowLimit_X2[3]+1;
       #DevState.DevState.DevState.staticDevState3[#statiDevStateMove_X2[3]] := #devStateHmi_X2[#staticCntState];
   END_IF;
   IF #_w3 AND (0 <> #staticCntLowLimit_X1[3]) THEN
       #statiDevStateMove_X2[3] := #staticCntState-#staticCntLowLimit_X2[3]+(#staticCntHighLimit_X1[3]-#staticCntLowLimit_X1[3]+2);
       #DevState.DevState.DevState.staticDevState3[#statiDevStateMove_X2[3]] := #devStateHmi_X2[#staticCntState];
   END_IF;
   #_w4 := (#staticCntState >= #staticCntLowLimit_X2[4]) AND (#staticCntState <= #staticCntHighLimit_X2[4]);
   IF #_w4 AND (0 = #staticCntLowLimit_X1[4]) THEN
       #statiDevStateMove_X2[4] := #staticCntState-#staticCntLowLimit_X2[4]+1;
       #DevState.DevState.DevState.staticDevState4[#statiDevStateMove_X2[4]] := #devStateHmi_X2[#staticCntState];
   END_IF;
   IF #_w4 AND (0 <> #staticCntLowLimit_X1[4]) THEN
       #statiDevStateMove_X2[4] := #staticCntState-#staticCntLowLimit_X2[4]+(#staticCntHighLimit_X1[4]-#staticCntLowLimit_X1[4]+2);
       #DevState.DevState.DevState.staticDevState4[#statiDevStateMove_X2[4]] := #devStateHmi_X2[#staticCntState];
   END_IF;
   #_w5 := (#staticCntState >= #staticCntLowLimit_X2[5]) AND (#staticCntState <= #staticCntHighLimit_X2[5]);
   IF #_w5 AND (0 = #staticCntLowLimit_X1[5]) THEN
       #statiDevStateMove_X2[5] := #staticCntState-#staticCntLowLimit_X2[5]+1;
       #DevState.DevState.DevState.staticDevState5[#statiDevStateMove_X2[5]] := #devStateHmi_X2[#staticCntState];
   END_IF;
   IF #_w5 AND (0 <> #staticCntLowLimit_X1[5]) THEN
       #statiDevStateMove_X2[5] := #staticCntState-#staticCntLowLimit_X2[5]+(#staticCntHighLimit_X1[5]-#staticCntLowLimit_X1[5]+2);
       #DevState.DevState.DevState.staticDevState5[#statiDevStateMove_X2[5]] := #devStateHmi_X2[#staticCntState];
   END_IF;
   #_w6 := (#staticCntState >= #staticCntLowLimit_X2[6]) AND (#staticCntState <= #staticCntHighLimit_X2[6]);
   IF #_w6 AND (0 = #staticCntLowLimit_X1[6]) THEN
       #statiDevStateMove_X2[6] := #staticCntState-#staticCntLowLimit_X2[6]+1;
       #DevState.DevState.DevState.staticDevState6[#statiDevStateMove_X2[6]] := #devStateHmi_X2[#staticCntState];
   END_IF;
   IF #_w6 AND (0 <> #staticCntLowLimit_X1[6]) THEN
       #statiDevStateMove_X2[6] := #staticCntState-#staticCntLowLimit_X2[6]+(#staticCntHighLimit_X1[6]-#staticCntLowLimit_X1[6]+2);
       #DevState.DevState.DevState.staticDevState6[#statiDevStateMove_X2[6]] := #devStateHmi_X2[#staticCntState];
   END_IF;
   #_w7 := (#staticCntState >= #staticCntLowLimit_X2[7]) AND (#staticCntState <= #staticCntHighLimit_X2[7]);
   IF #_w7 AND (0 = #staticCntLowLimit_X1[7]) THEN
       #statiDevStateMove_X2[7] := #staticCntState-#staticCntLowLimit_X2[7]+1;
       #DevState.DevState.DevState.staticDevState7[#statiDevStateMove_X2[7]] := #devStateHmi_X2[#staticCntState];
   END_IF;
   IF #_w7 AND (0 <> #staticCntLowLimit_X1[7]) THEN
       #statiDevStateMove_X2[7] := #staticCntState-#staticCntLowLimit_X2[7]+(#staticCntHighLimit_X1[7]-#staticCntLowLimit_X1[7]+2);
       #DevState.DevState.DevState.staticDevState7[#statiDevStateMove_X2[7]] := #devStateHmi_X2[#staticCntState];
   END_IF;
   #_w8 := (#staticCntState >= #staticCntLowLimit_X2[8]) AND (#staticCntState <= #staticCntHighLimit_X2[8]);
   #_w9 := #_w8 AND (0 = #staticCntLowLimit_X1[8]);
   IF #_w9 THEN
       #statiDevStateMove_X2[8] := #staticCntState-#staticCntLowLimit_X2[8]+1;
       #DevState.DevState.DevState.staticDevState8[#statiDevStateMove_X2[8]] := #devStateHmi_X2[#staticCntState];
   END_IF;
   #DevState.DigState[15] := #_w9;
   IF #_w8 AND (0 <> #staticCntLowLimit_X1[8]) THEN
       #statiDevStateMove_X2[8] := #staticCntState-#staticCntLowLimit_X2[8]+(#staticCntHighLimit_X1[8]-#staticCntLowLimit_X1[8]+2);
       #DevState.DevState.DevState.staticDevState8[#statiDevStateMove_X2[8]] := #devStateHmi_X2[#staticCntState];
   END_IF;
   #_w10 := (#staticCntState >= #staticCntLowLimit_X2[9]) AND (#staticCntState <= #staticCntHighLimit_X2[9]);
   IF #_w10 AND (0 = #staticCntLowLimit_X1[9]) THEN
       #statiDevStateMove_X2[9] := #staticCntState-#staticCntLowLimit_X2[9]+1;
       #DevState.DevState.DevState.staticDevState9[#statiDevStateMove_X2[9]] := #devStateHmi_X2[#staticCntState];
   END_IF;
   IF #_w10 AND (0 <> #staticCntLowLimit_X1[9]) THEN
       #statiDevStateMove_X2[9] := #staticCntState-#staticCntLowLimit_X2[9]+(#staticCntHighLimit_X1[9]-#staticCntLowLimit_X1[9]+2);
       #DevState.DevState.DevState.staticDevState9[#statiDevStateMove_X2[9]] := #devStateHmi_X2[#staticCntState];
   END_IF;
   #_w11 := (#staticCntState >= #staticCntLowLimit_X2[10]) AND (#staticCntState <= #staticCntHighLimit_X2[10]);
   IF #_w11 AND (0 = #staticCntLowLimit_X1[10]) THEN
       #statiDevStateMove_X2[10] := #staticCntState-#staticCntLowLimit_X2[10]+1;
       #DevState.DevState.DevState.staticDevState10[#statiDevStateMove_X2[10]] := #devStateHmi_X2[#staticCntState];
   END_IF;
   IF #_w11 AND (0 <> #staticCntLowLimit_X1[10]) THEN
       #statiDevStateMove_X2[10] := #staticCntState-#staticCntLowLimit_X2[10]+(#staticCntHighLimit_X1[10]-#staticCntLowLimit_X1[10]+2);
       #DevState.DevState.DevState.staticDevState10[#statiDevStateMove_X2[10]] := #devStateHmi_X2[#staticCntState];
   END_IF;
   #_w12 := (#staticCntState >= #staticCntLowLimit_X2[11]) AND (#staticCntState <= #staticCntHighLimit_X2[11]);
   IF #_w12 AND (0 = #staticCntLowLimit_X1[11]) THEN
       #statiDevStateMove_X2[11] := #staticCntState-#staticCntLowLimit_X2[11]+1;
       #DevState.DevState.DevState.staticDevState11[#statiDevStateMove_X2[11]] := #devStateHmi_X2[#staticCntState];
   END_IF;
   IF #_w12 AND (0 <> #staticCntLowLimit_X1[11]) THEN
       #statiDevStateMove_X2[11] := #staticCntState-#staticCntLowLimit_X2[11]+(#staticCntHighLimit_X1[11]-#staticCntLowLimit_X1[11]+2);
       #DevState.DevState.DevState.staticDevState11[#statiDevStateMove_X2[11]] := #devStateHmi_X2[#staticCntState];
   END_IF;
   #_w13 := (#staticCntState >= #staticCntLowLimit_X2[12]) AND (#staticCntState <= #staticCntHighLimit_X2[12]);
   IF #_w13 AND (0 = #staticCntLowLimit_X1[12]) THEN
       #statiDevStateMove_X2[12] := #staticCntState-#staticCntLowLimit_X2[12]+1;
       #DevState.DevState.DevState.staticDevState12[#statiDevStateMove_X2[12]] := #devStateHmi_X2[#staticCntState];
   END_IF;
   IF #_w13 AND (0 <> #staticCntLowLimit_X1[12]) THEN
       #statiDevStateMove_X2[12] := #staticCntState-#staticCntLowLimit_X2[12]+(#staticCntHighLimit_X1[12]-#staticCntLowLimit_X1[12]+2);
       #DevState.DevState.DevState.staticDevState12[#statiDevStateMove_X2[12]] := #devStateHmi_X2[#staticCntState];
   END_IF;
   #_w14 := (#staticCntState >= #staticCntLowLimit_X2[13]) AND (#staticCntState <= #staticCntHighLimit_X2[13]);
   IF #_w14 AND (0 = #staticCntLowLimit_X1[13]) THEN
       #statiDevStateMove_X2[13] := #staticCntState-#staticCntLowLimit_X2[13]+1;
       #DevState.DevState.DevState.staticDevState13[#statiDevStateMove_X2[13]] := #devStateHmi_X2[#staticCntState];
   END_IF;
   IF #_w14 AND (0 <> #staticCntLowLimit_X1[13]) THEN
       #statiDevStateMove_X2[13] := #staticCntState-#staticCntLowLimit_X2[13]+(#staticCntHighLimit_X1[13]-#staticCntLowLimit_X1[13]+2);
       #DevState.DevState.DevState.staticDevState13[#statiDevStateMove_X2[13]] := #devStateHmi_X2[#staticCntState];
   END_IF;
   #_w15 := (#staticCntState >= #staticCntLowLimit_X2[14]) AND (#staticCntState <= #staticCntHighLimit_X2[14]);
   IF #_w15 AND (0 = #staticCntLowLimit_X1[14]) THEN
       #statiDevStateMove_X2[14] := #staticCntState-#staticCntLowLimit_X2[14]+1;
       #DevState.DevState.DevState.staticDevState14[#statiDevStateMove_X2[14]] := #devStateHmi_X2[#staticCntState];
   END_IF;
   IF #_w15 AND (0 <> #staticCntLowLimit_X1[14]) THEN
       #statiDevStateMove_X2[14] := #staticCntState-#staticCntLowLimit_X2[14]+(#staticCntHighLimit_X1[14]-#staticCntLowLimit_X1[14]+2);
       #DevState.DevState.DevState.staticDevState14[#statiDevStateMove_X2[14]] := #devStateHmi_X2[#staticCntState];
   END_IF;
   #_w16 := (#staticCntState >= #staticCntLowLimit_X2[15]) AND (#staticCntState <= #staticCntHighLimit_X2[15]);
   IF #_w16 AND (0 = #staticCntLowLimit_X1[15]) THEN
       #statiDevStateMove_X2[15] := #staticCntState-#staticCntLowLimit_X2[15]+1;
       #DevState.DevState.DevState.staticDevState15[#statiDevStateMove_X2[15]] := #devStateHmi_X2[#staticCntState];
   END_IF;
   IF #_w16 AND (0 <> #staticCntLowLimit_X1[15]) THEN
       #statiDevStateMove_X2[15] := #staticCntState-#staticCntLowLimit_X2[15]+(#staticCntHighLimit_X1[15]-#staticCntLowLimit_X1[15]+2);
       #DevState.DevState.DevState.staticDevState15[#statiDevStateMove_X2[15]] := #devStateHmi_X2[#staticCntState];
   END_IF;
END_REGION

REGION Network 5 (SCL)
   IF #staticCntDev >= 16 THEN
       #staticCntDev := 1;

   ELSIF #staticCntDev < 16 THEN
       #DevState.DigState[#staticCntDev] := 0;
       IF #staticCntLowLimit_X2[#staticCntDev] <> 0 AND #staticCntHighLimit_X2[#staticCntDev] <> 0 THEN

           FOR #staticCntModuleState := #staticCntLowLimit_X2[#staticCntDev] TO #staticCntHighLimit_X2[#staticCntDev] DO
               #DevState.DigState[#staticCntDev] := #DevState.DigState[#staticCntDev] OR (#nomal <> #devStateHmi_X2[#staticCntModuleState].devStateBitCoded);
           END_FOR;

       END_IF;
       IF #staticCntLowLimit_X1[#staticCntDev] <> 0 AND #staticCntHighLimit_X1[#staticCntDev] <> 0 THEN

           FOR #staticCntModuleState := #staticCntLowLimit_X1[#staticCntDev] TO #staticCntHighLimit_X1[#staticCntDev] DO
               #DevState.DigState[#staticCntDev] := #DevState.DigState[#staticCntDev] OR (#nomal <> #devStateHmi_X1[#staticCntModuleState].devStateBitCoded);
           END_FOR;

       END_IF;
       #staticCntDev += 1;
   END_IF;
END_REGION

REGION Network 6
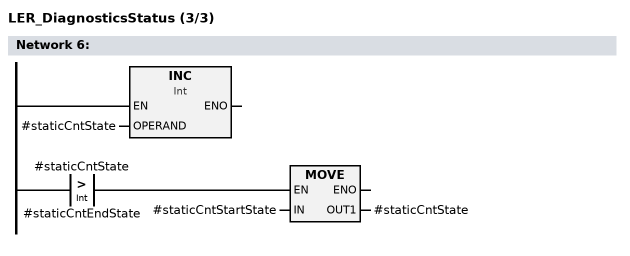
   RUNG wire#powerrail
      { S7_Templates := "DestType := Int" } Inc( #staticCntState )
   END_RUNG
   RUNG wire#powerrail
      { S7_Templates := "SrcType := Int" } GT_Contact(in1 := #staticCntState, in2 := #staticCntEndState)
      Move(in := #staticCntStartState, out1 => #staticCntState)
   END_RUNG
   // the same network as SCL:
   #staticCntState := #staticCntState + 1;
   IF #staticCntState > #staticCntEndState THEN #staticCntState := #staticCntStartState; END_IF;
END_REGION
END_FUNCTION_BLOCK
